// TwinCAT 3 PLC project DCSv1
// ProgramVersion: 3.1.4023.0
// libraries:
//   Tc2_MC2, * (Beckhoff Automation GmbH)
//   Tc2_MC2_Drive, * (Beckhoff Automation GmbH)
//   Tc2_SerialCom, * (Beckhoff Automation GmbH)
//   Tc2_Standard, * (Beckhoff Automation GmbH)
//   Tc2_System, * (Beckhoff Automation GmbH)
//   Tc2_Utilities, * (Beckhoff Automation GmbH)
//   Tc3_Module, * (Beckhoff Automation GmbH)
// project tree:
//   / ComTask.TcTTO, PlcTask.TcTTO
//   DUTs/DUTs/ arr8Bit.TcDUT
//   GVLs/GVLs/ GVL.TcGVL, GVL_IO.TcGVL (not stored), GVL_PN.TcGVL, GVL_RESD.TcGVL, GVL_ROB.TcGVL, ReadMe.TcGVL
//   POUs/Archive/ FB_Analog.TcPOU (not stored), P_ComEL6001.TcPOU (not stored)
//   POUs/Component/MIxer_Driver/ FB_Drive.TcPOU (not stored), FB_Mixer1_2.TcPOU
//   POUs/Component/ P_AP1_Check.TcPOU (not stored), P_AP1_OnOff.TcPOU (not stored), P_CC1_Enable.TcPOU (not stored), P_CP1_Check.TcPOU, P_CP1_Enable.TcPOU (not stored), P_MI1_OnOff.TcPOU (not stored), P_SP1_Check.TcPOU (not stored), P_SP1_OnOff.TcPOU (not stored)
//   POUs/Customed_Mode/ P_MI1_Curved_Speed.TcPOU (not stored)
//   POUs/ FB_GetOutputData.TcPOU, FB_Output_Speed.TcPOU (not stored), FB_SetConfigData.TcPOU (not stored), FB_SetOutputDataToIO.TcPOU, MAIN.TcPOU, P_Control_Mode.TcPOU, P_Manual_Operate.TcPOU (not stored), P_PNDataConvert.TcPOU, P_Robot_Operate.TcPOU, P_Laptop_Operate.TcPOU, temp.TcPOU
//   POUs/Utils/ F_Convert_2Byte_to_Uint.TcPOU, F_Convert_2Byte_to_Real.TcPOU, F_Convert_Bit_to_Byte.TcPOU, F_Convert_Uint_to_2Byte.TcPOU, F_LowpassFilter.TcPOU (not stored), F_Convert_2Byte_to_Int.TcPOU (not stored), F_Convert_Byte_to_Bit.TcPOU (not stored), F_Convert_Int_to_2Byte.TcPOU (not stored), F_DecimalData.TcPOU (not stored), F_Mapping.TcPOU (not stored), F_ScalAnalogOut.TcPOU
// real-time tasks:
//   TASK PlcTask: cycle T#10ms, priority 10, ADS port 350
//   TASK ComTask: cycle T#8ms, priority 5, ADS port 351
// motion (NC):
//   TASK NC-Task 1 SAF: cycle T#2ms, priority 4, ADS port 501
//   TASK NC-Task 1 SVB: cycle T#10ms, priority 8, ADS port 511
//   AXIS Mixer 1 (id 2)
//     General: UnitName=°, UnitFlags=#x00000004
//     Dynamic: Acceleration=7443.34, Deceleration=7443.34, Jerk=22330
//     Velo: RefSearch=49.6222741699219, RefSync=49.6222741699219, SlowManual=248.111370849609, FastManual=1488.66822509766, Fast=4962.22741699219, Maximum=4962.23
//     OtherSettings: AllowMotionCmdToSlave=true
//     encoder EncType=8
//       EncPara: ScaleFactorNumerator=45, ScaleFactorDenominator=1048576, Offset=-131121.7408, Inverse=true, MaxCount=#x007fffff, ReferenceSystem=2
//     drive DrvType=9
//       DrvPara: Inverse=true, MaxCount=#xffffffff, DriveControlDWord=#x00030100
//         Analog: VeloReferenz=5458.45015869141, VeloScale=1.02400649589962, ScaleFactorActTorque=0.1
//         TimeComp: TaskDelayCycles=1
//     controller CtrType=1
//       CtrPara: PriorControlFactor=1
//         Observer: BandWidth=20
//   AXIS Mixer 2 (id 3)
//     General: UnitName=°, UnitFlags=#x00000004
//     Dynamic: Acceleration=7443.34, Deceleration=7443.34, Jerk=22330
//     Velo: RefSearch=49.6222741699219, RefSync=49.6222741699219, SlowManual=248.111370849609, FastManual=1488.66822509766, Fast=4962.22741699219, Maximum=4962.23
//     OtherSettings: AllowMotionCmdToSlave=true
//     encoder EncType=8
//       EncPara: ScaleFactorNumerator=45, ScaleFactorDenominator=1048576, MaxCount=#x007fffff, ReferenceSystem=2
//     drive DrvType=9
//       DrvPara: MaxCount=#xffffffff, DriveControlDWord=#x00030100
//         Analog: VeloReferenz=5458.45015869141, VeloScale=1.02400649589962, ScaleFactorActTorque=0.1
//         TimeComp: TaskDelayCycles=1
//     controller CtrType=1
//       CtrPara: PriorControlFactor=1
//         Observer: BandWidth=20
// I/O:
//   DEVICE Device 1 (EtherCAT), AmsNetId 172.17.147.1.3.1
//     Term 1 (EK1200) [EK1200-5000 EtherCAT Power supply (2A E-Bus)]
//       Term 2 (EL1008) 30K3 [EL1008 8Ch. Dig. Input 24V, 3ms]
//       Term 3 (EL1008) 30K3.1 [EL1008 8Ch. Dig. Input 24V, 3ms]
//       Term 10 (EL1008) new [EL1008 8Ch. Dig. Input 24V, 3ms]
//       Term 4 (EL2008) 30K4 [EL2008 8Ch. Dig. Output 24V, 0.5A]
//       Term 5 (EL2008) 30K5 [EL2008 8Ch. Dig. Output 24V, 0.5A]
//       Term 12 (EL2008) new [EL2008 8Ch. Dig. Output 24V, 0.5A]
//       Term 13 (EL3022) new [EL3022 2Ch. Ana. Input 4-20mA DIFF]
//       Term 14 (EL3202) new [EL3202 2Ch. Ana. Input PT100 (RTD)]
//       Term 16 (EL3202) new pt100 [EL3202 2Ch. Ana. Input PT100 (RTD)]
//       Term 6 (EL3255) 30K5.1 [EL3255 5Ch. potentiometer measurement with sensor supply]
//       Term 7 (EL4134) 30K6 [EL4134 4Ch. Ana. Output -10/+10V, 16bit]
//       Term 8 (EL6001) [EL6001 Interface (RS232)]
//       Term 15 (EL6631-0010) [EL6631-0010 PROFINET IO Device]
//       Term 17 (EL6631) [EL6631 PROFINET IO Controller]
//       Term 9 (EL9011) [EL9011 End Terminal]
//   DEVICE Device 4 (EtherCAT), AmsNetId 172.17.147.1.5.1
//     Drive 11 (AX5206-0000-0213) [AX5206-0000-0213 EtherCAT Drive (SoE, 2 Ch.)]
//   DEVICE Device 1 (EL6631-0010), AmsNetId 5.57.158.168.2.1
//     robotbasicio [ABB Robotics The robot controller's internal PROFINET IO device. 888-3]
//       modules: Term 1 (DAP Module), Term 2 (DI 256 bytes), Term 3 (DO 256 bytes)
// variable links:
//   NC-Task 1 SAF/Axes/Mixer 1 <-> Device 4 (EtherCAT)/Drive 11 (AX5206-0000-0213)
//     Drive/Inputs/In/nDataIn1 <-> AT 1/Following distance
//     Drive/Inputs/In/nDcOutputTime <-> InfoData/DcOutputShift
//     Drive/Inputs/In/nState1 <-> AT 1/Drive status word @bit 8
//     Drive/Inputs/In/nState2 <-> AT 1/Drive status word
//     Drive/Inputs/In/nState4 @bit 1 <-> WcState/InputToggle
//     Drive/Inputs/In/nState4 <-> WcState/WcState
//     Drive/Outputs/Out/nCtrl1 <-> MDT 1/Master control word @bit 8
//     Drive/Outputs/Out/nDataOut1 <-> MDT 1/Position command value
//     Enc/Inputs/In/nDataIn1 <-> AT 1/Position feedback 1 value
//     Enc/Inputs/In/nDcInputTime <-> InfoData/DcInputShift
//     Enc/Inputs/In/nState4 @bit 1 <-> WcState/InputToggle
//     Enc/Inputs/In/nState4 <-> WcState/WcState
//   NC-Task 1 SAF/Axes/Mixer 2 <-> Device 4 (EtherCAT)/Drive 11 (AX5206-0000-0213)
//     Drive/Inputs/In/nDataIn1 <-> AT 2/Following distance
//     Drive/Inputs/In/nDcOutputTime <-> InfoData/DcOutputShift
//     Drive/Inputs/In/nState1 <-> AT 2/Drive status word @bit 8
//     Drive/Inputs/In/nState2 <-> AT 2/Drive status word
//     Drive/Inputs/In/nState4 @bit 1 <-> WcState/InputToggle
//     Drive/Inputs/In/nState4 <-> WcState/WcState
//     Drive/Outputs/Out/nCtrl1 <-> MDT 2/Master control word @bit 8
//     Drive/Outputs/Out/nDataOut1 <-> MDT 2/Position command value
//     Enc/Inputs/In/nDataIn1 <-> AT 2/Position feedback 1 value
//     Enc/Inputs/In/nDcInputTime <-> InfoData/DcInputShift
//     Enc/Inputs/In/nState4 @bit 1 <-> WcState/InputToggle
//     Enc/Inputs/In/nState4 <-> WcState/WcState
//   DCSv1/DCSv1 Instance <-> Device 1 (EL6631-0010)/robotbasicio
//     PlcTask Inputs/GVL_PN.DO_From_ROB <-> API/Term 3 (DO 256 bytes)/Subterm 5 (DO 256 bytes)/Inputs/Output 0
//     PlcTask Inputs/GVL_PN.DO_From_ROB[{0..4}] <-> API/Term 3 (DO 256 bytes)/Subterm 5 (DO 256 bytes)/Inputs/Output {0..4}  (5 links)
//     PlcTask Inputs/GVL_PN.GO_From_ROB[100] <-> API/Term 3 (DO 256 bytes)/Subterm 5 (DO 256 bytes)/Inputs/Output 100
//     PlcTask Inputs/GVL_PN.GO_From_ROB[101] <-> API/Term 3 (DO 256 bytes)/Subterm 5 (DO 256 bytes)/Inputs/Output 101
//     PlcTask Inputs/GVL_PN.GO_From_ROB[102] <-> API/Term 3 (DO 256 bytes)/Subterm 5 (DO 256 bytes)/Inputs/Output 102
//     PlcTask Inputs/GVL_PN.GO_From_ROB[103] <-> API/Term 3 (DO 256 bytes)/Subterm 5 (DO 256 bytes)/Inputs/Output 103
//     PlcTask Inputs/GVL_PN.GO_From_ROB[104] <-> API/Term 3 (DO 256 bytes)/Subterm 5 (DO 256 bytes)/Inputs/Output 104
//     PlcTask Inputs/GVL_PN.GO_From_ROB[105] <-> API/Term 3 (DO 256 bytes)/Subterm 5 (DO 256 bytes)/Inputs/Output 105
//     PlcTask Inputs/GVL_PN.GO_From_ROB[32] <-> API/Term 3 (DO 256 bytes)/Subterm 5 (DO 256 bytes)/Inputs/Output 32
//     PlcTask Inputs/GVL_PN.GO_From_ROB[33] <-> API/Term 3 (DO 256 bytes)/Subterm 5 (DO 256 bytes)/Inputs/Output 33
//     PlcTask Inputs/GVL_PN.GO_From_ROB[47] <-> API/Term 3 (DO 256 bytes)/Subterm 5 (DO 256 bytes)/Inputs/Output 47
//     PlcTask Inputs/GVL_PN.GO_From_ROB[48] <-> API/Term 3 (DO 256 bytes)/Subterm 5 (DO 256 bytes)/Inputs/Output 48
//     PlcTask Inputs/GVL_PN.GO_From_ROB[62] <-> API/Term 3 (DO 256 bytes)/Subterm 5 (DO 256 bytes)/Inputs/Output 62
//     PlcTask Inputs/GVL_PN.GO_From_ROB[63] <-> API/Term 3 (DO 256 bytes)/Subterm 5 (DO 256 bytes)/Inputs/Output 63
//     PlcTask Inputs/GVL_PN.GO_From_ROB[64] <-> API/Term 3 (DO 256 bytes)/Subterm 5 (DO 256 bytes)/Inputs/Output 64
//     PlcTask Inputs/GVL_PN.GO_From_ROB[65] <-> API/Term 3 (DO 256 bytes)/Subterm 5 (DO 256 bytes)/Inputs/Output 65
//     PlcTask Inputs/GVL_PN.GO_From_ROB[66] <-> API/Term 3 (DO 256 bytes)/Subterm 5 (DO 256 bytes)/Inputs/Output 66
//     PlcTask Inputs/GVL_PN.GO_From_ROB[67] <-> API/Term 3 (DO 256 bytes)/Subterm 5 (DO 256 bytes)/Inputs/Output 67
//     PlcTask Inputs/GVL_PN.GO_From_ROB[68] <-> API/Term 3 (DO 256 bytes)/Subterm 5 (DO 256 bytes)/Inputs/Output 68
//     PlcTask Inputs/GVL_PN.GO_From_ROB[69] <-> API/Term 3 (DO 256 bytes)/Subterm 5 (DO 256 bytes)/Inputs/Output 69
//     PlcTask Inputs/GVL_PN.GO_From_ROB[70] <-> API/Term 3 (DO 256 bytes)/Subterm 5 (DO 256 bytes)/Inputs/Output 70
//     PlcTask Inputs/GVL_PN.GO_From_ROB[71] <-> API/Term 3 (DO 256 bytes)/Subterm 5 (DO 256 bytes)/Inputs/Output 71
//     PlcTask Inputs/GVL_PN.GO_From_ROB[72] <-> API/Term 3 (DO 256 bytes)/Subterm 5 (DO 256 bytes)/Inputs/Output 72
//     PlcTask Inputs/GVL_PN.GO_From_ROB[73] <-> API/Term 3 (DO 256 bytes)/Subterm 5 (DO 256 bytes)/Inputs/Output 73
//     PlcTask Inputs/GVL_PN.GO_From_ROB[74] <-> API/Term 3 (DO 256 bytes)/Subterm 5 (DO 256 bytes)/Inputs/Output 74
//     PlcTask Inputs/GVL_PN.GO_From_ROB[75] <-> API/Term 3 (DO 256 bytes)/Subterm 5 (DO 256 bytes)/Inputs/Output 75
//     PlcTask Inputs/GVL_PN.GO_From_ROB[78] <-> API/Term 3 (DO 256 bytes)/Subterm 5 (DO 256 bytes)/Inputs/Output 78
//     PlcTask Inputs/GVL_PN.GO_From_ROB[79] <-> API/Term 3 (DO 256 bytes)/Subterm 5 (DO 256 bytes)/Inputs/Output 79
//     PlcTask Inputs/GVL_PN.GO_From_ROB[80] <-> API/Term 3 (DO 256 bytes)/Subterm 5 (DO 256 bytes)/Inputs/Output 80
//     PlcTask Inputs/GVL_PN.GO_From_ROB[81] <-> API/Term 3 (DO 256 bytes)/Subterm 5 (DO 256 bytes)/Inputs/Output 81
//     PlcTask Inputs/GVL_PN.GO_From_ROB[82] <-> API/Term 3 (DO 256 bytes)/Subterm 5 (DO 256 bytes)/Inputs/Output 82
//     PlcTask Inputs/GVL_PN.GO_From_ROB[83] <-> API/Term 3 (DO 256 bytes)/Subterm 5 (DO 256 bytes)/Inputs/Output 83
//     PlcTask Inputs/GVL_PN.GO_From_ROB[84] <-> API/Term 3 (DO 256 bytes)/Subterm 5 (DO 256 bytes)/Inputs/Output 84
//     PlcTask Inputs/GVL_PN.GO_From_ROB[85] <-> API/Term 3 (DO 256 bytes)/Subterm 5 (DO 256 bytes)/Inputs/Output 85
//     PlcTask Inputs/GVL_PN.GO_From_ROB[86] <-> API/Term 3 (DO 256 bytes)/Subterm 5 (DO 256 bytes)/Inputs/Output 86
//     PlcTask Inputs/GVL_PN.GO_From_ROB[87] <-> API/Term 3 (DO 256 bytes)/Subterm 5 (DO 256 bytes)/Inputs/Output 87
//     PlcTask Inputs/GVL_PN.GO_From_ROB[88] <-> API/Term 3 (DO 256 bytes)/Subterm 5 (DO 256 bytes)/Inputs/Output 88
//     PlcTask Inputs/GVL_PN.GO_From_ROB[89] <-> API/Term 3 (DO 256 bytes)/Subterm 5 (DO 256 bytes)/Inputs/Output 89
//     PlcTask Inputs/GVL_PN.GO_From_ROB[90] <-> API/Term 3 (DO 256 bytes)/Subterm 5 (DO 256 bytes)/Inputs/Output 90
//     PlcTask Inputs/GVL_PN.GO_From_ROB[91] <-> API/Term 3 (DO 256 bytes)/Subterm 5 (DO 256 bytes)/Inputs/Output 91
//     PlcTask Inputs/GVL_PN.GO_From_ROB[94] <-> API/Term 3 (DO 256 bytes)/Subterm 5 (DO 256 bytes)/Inputs/Output 94
//     PlcTask Inputs/GVL_PN.GO_From_ROB[95] <-> API/Term 3 (DO 256 bytes)/Subterm 5 (DO 256 bytes)/Inputs/Output 95
//     PlcTask Inputs/GVL_PN.GO_From_ROB[96] <-> API/Term 3 (DO 256 bytes)/Subterm 5 (DO 256 bytes)/Inputs/Output 96
//     PlcTask Inputs/GVL_PN.GO_From_ROB[97] <-> API/Term 3 (DO 256 bytes)/Subterm 5 (DO 256 bytes)/Inputs/Output 97
//     PlcTask Inputs/GVL_PN.GO_From_ROB[98] <-> API/Term 3 (DO 256 bytes)/Subterm 5 (DO 256 bytes)/Inputs/Output 98
//     PlcTask Inputs/GVL_PN.GO_From_ROB[99] <-> API/Term 3 (DO 256 bytes)/Subterm 5 (DO 256 bytes)/Inputs/Output 99
//     PlcTask Outputs/GVL_PN.DI_To_ROB[0]/data8Bit[0] <-> API/Term 2 (DI 256 bytes)/Subterm 4 (DI 256 bytes)/Outputs/Input 0[0]
//     PlcTask Outputs/GVL_PN.DI_To_ROB[0]/data8Bit[1] <-> API/Term 2 (DI 256 bytes)/Subterm 4 (DI 256 bytes)/Outputs/Input 0[1]
//     PlcTask Outputs/GVL_PN.DI_To_ROB[0]/data8Bit[2] <-> API/Term 2 (DI 256 bytes)/Subterm 4 (DI 256 bytes)/Outputs/Input 0[2]
//     PlcTask Outputs/GVL_PN.DI_To_ROB[0]/data8Bit[3] <-> API/Term 2 (DI 256 bytes)/Subterm 4 (DI 256 bytes)/Outputs/Input 0[3]
//     PlcTask Outputs/GVL_PN.DI_To_ROB[0]/data8Bit[4] <-> API/Term 2 (DI 256 bytes)/Subterm 4 (DI 256 bytes)/Outputs/Input 0[4]
//     PlcTask Outputs/GVL_PN.DI_To_ROB[0]/data8Bit[5] <-> API/Term 2 (DI 256 bytes)/Subterm 4 (DI 256 bytes)/Outputs/Input 0[5]
//     PlcTask Outputs/GVL_PN.DI_To_ROB[0]/data8Bit[6] <-> API/Term 2 (DI 256 bytes)/Subterm 4 (DI 256 bytes)/Outputs/Input 0[6]
//     PlcTask Outputs/GVL_PN.DI_To_ROB[0]/data8Bit[7] <-> API/Term 2 (DI 256 bytes)/Subterm 4 (DI 256 bytes)/Outputs/Input 0[7]
//     PlcTask Outputs/GVL_PN.DI_To_ROB[1]/data8Bit[0] <-> API/Term 2 (DI 256 bytes)/Subterm 4 (DI 256 bytes)/Outputs/Input 1[0]
//     PlcTask Outputs/GVL_PN.DI_To_ROB[1]/data8Bit[1] <-> API/Term 2 (DI 256 bytes)/Subterm 4 (DI 256 bytes)/Outputs/Input 1[1]
//     PlcTask Outputs/GVL_PN.DI_To_ROB[1]/data8Bit[2] <-> API/Term 2 (DI 256 bytes)/Subterm 4 (DI 256 bytes)/Outputs/Input 1[2]
//     PlcTask Outputs/GVL_PN.DI_To_ROB[1]/data8Bit[3] <-> API/Term 2 (DI 256 bytes)/Subterm 4 (DI 256 bytes)/Outputs/Input 1[3]
//     PlcTask Outputs/GVL_PN.DI_To_ROB[1]/data8Bit[4] <-> API/Term 2 (DI 256 bytes)/Subterm 4 (DI 256 bytes)/Outputs/Input 1[4]
//     PlcTask Outputs/GVL_PN.DI_To_ROB[1]/data8Bit[5] <-> API/Term 2 (DI 256 bytes)/Subterm 4 (DI 256 bytes)/Outputs/Input 1[5]
//     PlcTask Outputs/GVL_PN.DI_To_ROB[1]/data8Bit[6] <-> API/Term 2 (DI 256 bytes)/Subterm 4 (DI 256 bytes)/Outputs/Input 1[6]
//     PlcTask Outputs/GVL_PN.DI_To_ROB[1]/data8Bit[7] <-> API/Term 2 (DI 256 bytes)/Subterm 4 (DI 256 bytes)/Outputs/Input 1[7]
//     PlcTask Outputs/GVL_PN.DI_To_ROB[2]/data8Bit[0] <-> API/Term 2 (DI 256 bytes)/Subterm 4 (DI 256 bytes)/Outputs/Input 2[0]
//     PlcTask Outputs/GVL_PN.DI_To_ROB[2]/data8Bit[1] <-> API/Term 2 (DI 256 bytes)/Subterm 4 (DI 256 bytes)/Outputs/Input 2[1]
//     PlcTask Outputs/GVL_PN.DI_To_ROB[2]/data8Bit[2] <-> API/Term 2 (DI 256 bytes)/Subterm 4 (DI 256 bytes)/Outputs/Input 2[2]
//     PlcTask Outputs/GVL_PN.DI_To_ROB[2]/data8Bit[3] <-> API/Term 2 (DI 256 bytes)/Subterm 4 (DI 256 bytes)/Outputs/Input 2[3]
//     PlcTask Outputs/GVL_PN.DI_To_ROB[2]/data8Bit[4] <-> API/Term 2 (DI 256 bytes)/Subterm 4 (DI 256 bytes)/Outputs/Input 2[4]
//     PlcTask Outputs/GVL_PN.DI_To_ROB[2]/data8Bit[5] <-> API/Term 2 (DI 256 bytes)/Subterm 4 (DI 256 bytes)/Outputs/Input 2[5]
//     PlcTask Outputs/GVL_PN.DI_To_ROB[2]/data8Bit[6] <-> API/Term 2 (DI 256 bytes)/Subterm 4 (DI 256 bytes)/Outputs/Input 2[6]
//     PlcTask Outputs/GVL_PN.DI_To_ROB[2]/data8Bit[7] <-> API/Term 2 (DI 256 bytes)/Subterm 4 (DI 256 bytes)/Outputs/Input 2[7]
//     PlcTask Outputs/GVL_PN.DI_To_ROB[3]/data8Bit[0] <-> API/Term 2 (DI 256 bytes)/Subterm 4 (DI 256 bytes)/Outputs/Input 3[0]
//     PlcTask Outputs/GVL_PN.DI_To_ROB[3]/data8Bit[1] <-> API/Term 2 (DI 256 bytes)/Subterm 4 (DI 256 bytes)/Outputs/Input 3[1]
//     PlcTask Outputs/GVL_PN.DI_To_ROB[3]/data8Bit[2] <-> API/Term 2 (DI 256 bytes)/Subterm 4 (DI 256 bytes)/Outputs/Input 3[2]
//     PlcTask Outputs/GVL_PN.DI_To_ROB[3]/data8Bit[3] <-> API/Term 2 (DI 256 bytes)/Subterm 4 (DI 256 bytes)/Outputs/Input 3[3]
//     PlcTask Outputs/GVL_PN.DI_To_ROB[3]/data8Bit[4] <-> API/Term 2 (DI 256 bytes)/Subterm 4 (DI 256 bytes)/Outputs/Input 3[4]
//     PlcTask Outputs/GVL_PN.DI_To_ROB[3]/data8Bit[5] <-> API/Term 2 (DI 256 bytes)/Subterm 4 (DI 256 bytes)/Outputs/Input 3[5]
//     PlcTask Outputs/GVL_PN.DI_To_ROB[3]/data8Bit[6] <-> API/Term 2 (DI 256 bytes)/Subterm 4 (DI 256 bytes)/Outputs/Input 3[6]
//     PlcTask Outputs/GVL_PN.DI_To_ROB[3]/data8Bit[7] <-> API/Term 2 (DI 256 bytes)/Subterm 4 (DI 256 bytes)/Outputs/Input 3[7]
//     PlcTask Outputs/GVL_PN.DI_To_ROB[4]/data8Bit[0] <-> API/Term 2 (DI 256 bytes)/Subterm 4 (DI 256 bytes)/Outputs/Input 4[0]
//     PlcTask Outputs/GVL_PN.DI_To_ROB[4]/data8Bit[1] <-> API/Term 2 (DI 256 bytes)/Subterm 4 (DI 256 bytes)/Outputs/Input 4[1]
//     PlcTask Outputs/GVL_PN.DI_To_ROB[4]/data8Bit[2] <-> API/Term 2 (DI 256 bytes)/Subterm 4 (DI 256 bytes)/Outputs/Input 4[2]
//     PlcTask Outputs/GVL_PN.DI_To_ROB[4]/data8Bit[3] <-> API/Term 2 (DI 256 bytes)/Subterm 4 (DI 256 bytes)/Outputs/Input 4[3]
//     PlcTask Outputs/GVL_PN.DI_To_ROB[4]/data8Bit[4] <-> API/Term 2 (DI 256 bytes)/Subterm 4 (DI 256 bytes)/Outputs/Input 4[4]
//     PlcTask Outputs/GVL_PN.DI_To_ROB[4]/data8Bit[5] <-> API/Term 2 (DI 256 bytes)/Subterm 4 (DI 256 bytes)/Outputs/Input 4[5]
//     PlcTask Outputs/GVL_PN.DI_To_ROB[4]/data8Bit[6] <-> API/Term 2 (DI 256 bytes)/Subterm 4 (DI 256 bytes)/Outputs/Input 4[6]
//     PlcTask Outputs/GVL_PN.DI_To_ROB[4]/data8Bit[7] <-> API/Term 2 (DI 256 bytes)/Subterm 4 (DI 256 bytes)/Outputs/Input 4[7]
//     PlcTask Outputs/GVL_PN.GI_To_ROB[106] <-> API/Term 2 (DI 256 bytes)/Subterm 4 (DI 256 bytes)/Outputs/Input 106
//     PlcTask Outputs/GVL_PN.GI_To_ROB[107] <-> API/Term 2 (DI 256 bytes)/Subterm 4 (DI 256 bytes)/Outputs/Input 107
//     PlcTask Outputs/GVL_PN.GI_To_ROB[32] <-> API/Term 2 (DI 256 bytes)/Subterm 4 (DI 256 bytes)/Outputs/Input 32
//     PlcTask Outputs/GVL_PN.GI_To_ROB[33] <-> API/Term 2 (DI 256 bytes)/Subterm 4 (DI 256 bytes)/Outputs/Input 33
//     PlcTask Outputs/GVL_PN.GI_To_ROB[47] <-> API/Term 2 (DI 256 bytes)/Subterm 4 (DI 256 bytes)/Outputs/Input 47
//     PlcTask Outputs/GVL_PN.GI_To_ROB[48] <-> API/Term 2 (DI 256 bytes)/Subterm 4 (DI 256 bytes)/Outputs/Input 48
//     PlcTask Outputs/GVL_PN.GI_To_ROB[49] <-> API/Term 2 (DI 256 bytes)/Subterm 4 (DI 256 bytes)/Outputs/Input 49
//     PlcTask Outputs/GVL_PN.GI_To_ROB[50] <-> API/Term 2 (DI 256 bytes)/Subterm 4 (DI 256 bytes)/Outputs/Input 50
//     PlcTask Outputs/GVL_PN.GI_To_ROB[51] <-> API/Term 2 (DI 256 bytes)/Subterm 4 (DI 256 bytes)/Outputs/Input 51
//     PlcTask Outputs/GVL_PN.GI_To_ROB[52] <-> API/Term 2 (DI 256 bytes)/Subterm 4 (DI 256 bytes)/Outputs/Input 52
//     PlcTask Outputs/GVL_PN.GI_To_ROB[53] <-> API/Term 2 (DI 256 bytes)/Subterm 4 (DI 256 bytes)/Outputs/Input 53
//     PlcTask Outputs/GVL_PN.GI_To_ROB[54] <-> API/Term 2 (DI 256 bytes)/Subterm 4 (DI 256 bytes)/Outputs/Input 54
//     PlcTask Outputs/GVL_PN.GI_To_ROB[55] <-> API/Term 2 (DI 256 bytes)/Subterm 4 (DI 256 bytes)/Outputs/Input 55
//     PlcTask Outputs/GVL_PN.GI_To_ROB[56] <-> API/Term 2 (DI 256 bytes)/Subterm 4 (DI 256 bytes)/Outputs/Input 56
//     PlcTask Outputs/GVL_PN.GI_To_ROB[57] <-> API/Term 2 (DI 256 bytes)/Subterm 4 (DI 256 bytes)/Outputs/Input 57
//     PlcTask Outputs/GVL_PN.GI_To_ROB[58] <-> API/Term 2 (DI 256 bytes)/Subterm 4 (DI 256 bytes)/Outputs/Input 58
//     PlcTask Outputs/GVL_PN.GI_To_ROB[59] <-> API/Term 2 (DI 256 bytes)/Subterm 4 (DI 256 bytes)/Outputs/Input 59
//     PlcTask Outputs/GVL_PN.GI_To_ROB[60] <-> API/Term 2 (DI 256 bytes)/Subterm 4 (DI 256 bytes)/Outputs/Input 60
//     PlcTask Outputs/GVL_PN.GI_To_ROB[61] <-> API/Term 2 (DI 256 bytes)/Subterm 4 (DI 256 bytes)/Outputs/Input 61
//     PlcTask Outputs/GVL_PN.GI_To_ROB[62] <-> API/Term 2 (DI 256 bytes)/Subterm 4 (DI 256 bytes)/Outputs/Input 62
//     PlcTask Outputs/GVL_PN.GI_To_ROB[77] <-> API/Term 2 (DI 256 bytes)/Subterm 4 (DI 256 bytes)/Outputs/Input 77
//     PlcTask Outputs/GVL_PN.GI_To_ROB[78] <-> API/Term 2 (DI 256 bytes)/Subterm 4 (DI 256 bytes)/Outputs/Input 78
//     PlcTask Outputs/GVL_PN.GI_To_ROB[79] <-> API/Term 2 (DI 256 bytes)/Subterm 4 (DI 256 bytes)/Outputs/Input 79
//     PlcTask Outputs/GVL_PN.GI_To_ROB[80] <-> API/Term 2 (DI 256 bytes)/Subterm 4 (DI 256 bytes)/Outputs/Input 80
//     PlcTask Outputs/GVL_PN.GI_To_ROB[81] <-> API/Term 2 (DI 256 bytes)/Subterm 4 (DI 256 bytes)/Outputs/Input 81
//     PlcTask Outputs/GVL_PN.GI_To_ROB[82] <-> API/Term 2 (DI 256 bytes)/Subterm 4 (DI 256 bytes)/Outputs/Input 82
//     PlcTask Outputs/GVL_PN.GI_To_ROB[92] <-> API/Term 2 (DI 256 bytes)/Subterm 4 (DI 256 bytes)/Outputs/Input 92
//     PlcTask Outputs/GVL_PN.GI_To_ROB[93] <-> API/Term 2 (DI 256 bytes)/Subterm 4 (DI 256 bytes)/Outputs/Input 93
//   DCSv1/DCSv1 Instance <-> Device 1 (EtherCAT)/Term 1 (EK1200)/Term 10 (EL1008) new
//     PlcTask Inputs/GVL_IO.ib_SP1_No_Error <-> Channel 2/Input
//     PlcTask Inputs/GVL_IO.ib_SP1_Ready <-> Channel 1/Input
//   DCSv1/DCSv1 Instance <-> Device 1 (EtherCAT)/Term 1 (EK1200)/Term 13 (EL3022) new
//     PlcTask Inputs/GVL_IO.in_Pressure_Funnel <-> AI Standard Channel 1/Value
//     PlcTask Inputs/GVL_IO.in_Pressure_Pump <-> AI Standard Channel 2/Value
//   DCSv1/DCSv1 Instance <-> Device 1 (EtherCAT)/Term 1 (EK1200)/Term 14 (EL3202) new
//     PlcTask Inputs/GVL_IO.in_Temp_CPump <-> RTD Inputs Channel 2/Value
//     PlcTask Inputs/GVL_IO.in_Temp_CPump_fresh <-> RTD Inputs Channel 1/Value
//   DCSv1/DCSv1 Instance <-> Device 1 (EtherCAT)/Term 1 (EK1200)/Term 16 (EL3202) new pt100
//     PlcTask Inputs/GVL_IO.in_Temp_Funnel_Outlet <-> RTD Inputs Channel 2/Value
//   DCSv1/DCSv1 Instance <-> Device 1 (EtherCAT)/Term 1 (EK1200)/Term 2 (EL1008) 30K3
//     PlcTask Inputs/GVL_IO.ib_AP1_No_Error <-> Channel 6/Input
//     PlcTask Inputs/GVL_IO.ib_AP1_Ready <-> Channel 5/Input
//     PlcTask Inputs/GVL_IO.ib_CC1_Button_Mode_Laptop <-> Channel 8/Input
//     PlcTask Inputs/GVL_IO.ib_CC1_Button_Reset <-> Channel 7/Input
//     PlcTask Inputs/GVL_IO.ib_CC1_Safety_Ready <-> Channel 1/Input
//     PlcTask Inputs/GVL_IO.ib_CP1_Drive_Error <-> Channel 4/Input
//     PlcTask Inputs/GVL_IO.ib_CP1_Ready <-> Channel 3/Input
//     PlcTask Inputs/GVL_IO.ib_CP1_Safety_Grid_Mounted <-> Channel 2/Input
//   DCSv1/DCSv1 Instance <-> Device 1 (EtherCAT)/Term 1 (EK1200)/Term 3 (EL1008) 30K3.1
//     PlcTask Inputs/GVL_IO.ib_AP1_Button_Not_Off <-> Channel 7/Input
//     PlcTask Inputs/GVL_IO.ib_AP1_Button_On <-> Channel 6/Input
//     PlcTask Inputs/GVL_IO.ib_CC1_Button_Mode_Manual <-> Channel 1/Input
//     PlcTask Inputs/GVL_IO.ib_MI1_Button_Not_Off <-> Channel 3/Input
//     PlcTask Inputs/GVL_IO.ib_MI1_Button_On <-> Channel 2/Input
//     PlcTask Inputs/GVL_IO.ib_SP1_Button_Not_Off <-> Channel 5/Input
//     PlcTask Inputs/GVL_IO.ib_SP1_Button_On <-> Channel 4/Input
//   DCSv1/DCSv1 Instance <-> Device 1 (EtherCAT)/Term 1 (EK1200)/Term 4 (EL2008) 30K4
//     PlcTask Outputs/GVL_IO.ob_AP1_Pressure_Ok <-> Channel 7/Output
//     PlcTask Outputs/GVL_IO.ob_AP1_Pulse <-> Channel 8/Output
//     PlcTask Outputs/GVL_IO.ob_AP1_Start <-> Channel 6/Output
//     PlcTask Outputs/GVL_IO.ob_CC1_Safety_Reset <-> Channel 1/Output
//     PlcTask Outputs/GVL_IO.ob_CP1_Backward <-> Channel 5/Output
//     PlcTask Outputs/GVL_IO.ob_CP1_Forward <-> Channel 4/Output
//     PlcTask Outputs/GVL_IO.ob_CP1_Start <-> Channel 3/Output
//     PlcTask Outputs/GVL_IO.ob_CP1_Stop <-> Channel 2/Output
//   DCSv1/DCSv1 Instance <-> Device 1 (EtherCAT)/Term 1 (EK1200)/Term 5 (EL2008) 30K5
//     PlcTask Outputs/GVL_IO.ob_AP1_Not_Empty <-> Channel 1/Output
//     PlcTask Outputs/GVL_IO.ob_AP1_Power_On <-> Channel 2/Output
//     PlcTask Outputs/GVL_IO.ob_SP1_Not_Empty <-> Channel 6/Output
//     PlcTask Outputs/GVL_IO.ob_SP1_Power_On <-> Channel 7/Output
//     PlcTask Outputs/GVL_IO.ob_SP1_Pressure_Ok <-> Channel 4/Output
//     PlcTask Outputs/GVL_IO.ob_SP1_Pulse <-> Channel 5/Output
//     PlcTask Outputs/GVL_IO.ob_SP1_Start <-> Channel 3/Output
//   DCSv1/DCSv1 Instance <-> Device 1 (EtherCAT)/Term 1 (EK1200)/Term 6 (EL3255) 30K5.1
//     PlcTask Inputs/GVL.nInputSpare1 <-> AI Standard Channel 4/Value
//     PlcTask Inputs/GVL.nInputSpare2 <-> AI Standard Channel 5/Value
//     PlcTask Inputs/GVL_IO.in_AP1_Poti_Speed <-> AI Standard Channel 3/Value
//     PlcTask Inputs/GVL_IO.in_MI1_Poti_Speed <-> AI Standard Channel 1/Value
//   DCSv1/DCSv1 Instance <-> Device 1 (EtherCAT)/Term 1 (EK1200)/Term 7 (EL4134) 30K6
//     PlcTask Outputs/GVL_IO.on_AP1_Speed <-> AO Output Channel 2/Analog output
//     PlcTask Outputs/GVL_IO.on_CP1_Speed <-> AO Output Channel 1/Analog output
//     PlcTask Outputs/GVL_IO.on_SP1_Speed <-> AO Output Channel 3/Analog output
//   DCSv1/DCSv1 Instance <-> Device 1 (EtherCAT)/Term 1 (EK1200)/Term 8 (EL6001)
//     ComTask Inputs/GVL.stIn_EL6001/D <-> COM Inputs/Data In 0
//     ComTask Inputs/GVL.stIn_EL6001/D @bit {8..168 step 8} <-> COM Inputs/Data In {1..21}  (21 links)
//     ComTask Inputs/GVL.stIn_EL6001/Status <-> COM Inputs/Status
//     ComTask Outputs/GVL.stOut_EL6001/Ctrl <-> COM Outputs/Ctrl
//     ComTask Outputs/GVL.stOut_EL6001/D <-> COM Outputs/Data Out 0
//     ComTask Outputs/GVL.stOut_EL6001/D @bit {8..168 step 8} <-> COM Outputs/Data Out {1..21}  (21 links)
//   DCSv1/DCSv1 Instance <-> Device 4 (EtherCAT)/Drive 11 (AX5206-0000-0213)
//     PlcTask Inputs/GVL_IO.in_MID1_ActAbsCurrent <-> AT 1/Actual absolute current
//     PlcTask Inputs/GVL_IO.in_MID2_ActAbsCurrent <-> AT 2/Actual absolute current
//     PlcTask Inputs/GVL_IO.in_MID1_ActMotorTemperature <-> AT 1/Motor temperature
//     PlcTask Inputs/GVL_IO.in_MID2_ActMotorTemperature <-> AT 2/Motor temperature
//   DCSv1/DCSv1 Instance <-> NC-Task 1 SAF/Axes/Mixer 1
//     PlcTask Inputs/GVL.Axis_Mixer1.NcToPlc <-> Outputs/ToPlc
//     PlcTask Outputs/GVL.Axis_Mixer1.PlcToNc <-> Inputs/FromPlc
//   DCSv1/DCSv1 Instance <-> NC-Task 1 SAF/Axes/Mixer 2
//     PlcTask Inputs/GVL.Axis_Mixer2.NcToPlc <-> Outputs/ToPlc
//     PlcTask Outputs/GVL.Axis_Mixer2.PlcToNc <-> Inputs/FromPlc

CONFIGURATION DCSv1
    RESOURCE PLC ON TwinCAT3
        TASK ComTask(INTERVAL := T#8ms, PRIORITY := 5);
        TASK PlcTask(INTERVAL := T#10ms, PRIORITY := 10);
        PROGRAM P_ComEL6001 WITH ComTask : P_ComEL6001;
        PROGRAM MAIN WITH PlcTask : MAIN;
    END_RESOURCE
END_CONFIGURATION

// ---- DUTs/DUTs/arr8Bit.TcDUT
TYPE arr8Bit :
STRUCT
	data8Bit : ARRAY[0..7] OF BOOL;
END_STRUCT
END_TYPE

// ---- GVLs/GVLs/GVL.TcGVL
{attribute 'qualified_only'}
// ***********************************************************************************
//
// Müller-steinag Gruppe, Kandergrien Einigen, CH-3646 Bern
// ETH Zurich, Building HIF E26, Laura-Hezner-Weg 7, CH-8093 Zürich
// 
// ***********************************************************************************
// 
// PROJECT     :  A061 Digital Casting System 
// FUNCTION    :  Global Varable Decelerate
// AUTHOR      :  Weiting Chen
// EMAIL       :  chenw@usi.ch
// Copyright   :  USI Mendrisio; ETH Zürich; Müller-steinag Gruppe (CH) 2023
// Contributor :  Mathias Suter/ Philippe Fleischmann
//
// ***********************************************************************************

VAR_GLOBAL
	
    // get
	//
	// Concrete Controller 1
	b_mode_manual : BOOL;
	b_mode_laptop : BOOL; 
	b_mode_robot : BOOL;  
	
	b_CC1_enable :BOOL;
	b_CC1_power_on: BOOL;
	s_current_mode: STRING;
	
	//
	// Mixer 1
	b_MI1_ReadToDrive : BOOL;
	b_MI1_Is_Run : BOOL;
	
	f_MI1_MaxSpeed : REAL := 720 ; //distance/s] (equel to 120 rpm, by measurement 221006)
	n_MI1_OverrideSpeed :INT;
	b_Ml1_Enable : BOOL;
	b_Ml1_Set_Run : BOOL;
	
	f_MI1_ActSpeedM1 : INT;
	f_MI1_ActSpeedM2 : INT;
	
	// Data Communication Axis Mixers
	// Mixer drive A 
	Axis_Mixer1: AXIS_REF;
	
	f_MID1_ActCurrent:REAL;
	f_MID1_ActTorque:REAL;
	
	//
	// Mixer drive B
	Axis_Mixer2: AXIS_REF;
	f_MID2_ActCurrent:REAL;
	f_MID2_ActTorque:REAL;
	
	//
	// Concrete Pump 1
	b_CP1_Check_On : BOOL; //??
	b_CP1_is_run : BOOL;
	b_CP1_is_ready : BOOL;	
	b_CP1_power_on :BOOL;
	b_CP1_safety_grid_on : BOOL;
	b_CP1_drive_error :BOOL;
	
	//
	// Admixture pump 1 (High dosage)
	b_AP1_Is_Run : BOOL;
	b_AP1_Check_On : BOOL;
	b_AP1_is_ready : BOOL;
	b_AP1_no_error : BOOL;
	
	//f_AP1_Override : LREAL; 
	
	//
	// Spare Admixture pump 1 (Low dosage)
	b_SP1_Is_Run : BOOL;
	b_SP1_Check_On : BOOL;
	b_SP1_is_ready : BOOL;
	b_SP1_no_error : BOOL;
	
	//f_SP1_Override :LREAL;

	// Config
	// Concrete Pump 1
	f_CP1_Max_Flowrate : REAL;
	f_CP1_Check_Flowrate : REAL;
	t_CP1_Check_Duration : TIME;
 	n_CP1_Flush_Flowrate :REAL;
	
	// Admixture pump (High)
	n_AP1_Max_Flowrate : REAL;
	n_AP1_Check_Flowrate : REAL;
	t_AP1_Check_Duration : TIME;
	n_AP1_Flush_Flowrate : REAL;
	f_AP1_Check_Mass : REAL;
	
	// Admixture pump (low)
	n_SP1_Max_Flowrate : REAL;
	n_SP1_Check_Flowrate : REAL;
	t_SP1_Check_Duration : TIME;
	n_SP1_Flush_Flowrate : REAL;
	f_SP1_Check_Mass : REAL;
	
	
	
	
	
	// 
	// Data Communication RS-232 (Spare)
	TxBufferEL								: ComBuffer;
	RxBufferEL								: ComBuffer;
	
			

	//
	// Control Input Speed
	fControlMixerPumpSpeed					: REAL; 
	fControlPeristalticPumpSpeed			: REAL; 
	fControlDosingPumpSpeed					: REAL; 
	fInputSpare1							: REAL; 
	fInputSpare2							: REAL; 
	
	//
	// Output Speed
	fConcretePumpSpeed						: REAL;
	fDosingPumpSpeed						: REAL;
	fOutputSpare1							: REAL;
	fOutputSpare2							: REAL;
	
	
	//
	//Hardware Input
	bSafetyIO						AT %I*	: BOOL;
	// bConcretePumpSafetyGridMounted	AT %I*	: BOOL;
	// bConcretePumpReady				AT %I*	: BOOL;
	// bConcretePumpFcError				AT %I*	: BOOL;
	bDosingPumpReady				AT %I*	: BOOL;
	bDosingPumpNoError				AT %I*	: BOOL;
	bControlResetSafety				AT %I*	: BOOL;
	bControlLaptop					AT %I*	: BOOL;
	bControlManual					AT %I*	: BOOL;	
	nControlMixerPumpOn				AT %I*	: BOOL; 
	nControlMixerPumpOff			AT %I*	: BOOL; 
	nControlConcretPumpOn			AT %I*	: BOOL; 
	nControlConcretPumpOff			AT %I*	: BOOL; 
	nControlDosingPumpOn			AT %I*	: BOOL; 
	nControlDosingPumpOff			AT %I*	: BOOL; 
	bInputSpare1					AT %I*	: BOOL;
		
	nControlMixerPumpSpeed			AT %I*	: INT; 
	// nControlPeristalticPumpSpeed	AT %I*	: INT; 
	nControlDosingPumpSpeed			AT %I*	: INT; 
	nInputSpare1					AT %I*	: INT; 
	nInputSpare2					AT %I*	: INT; 

	
	//
	//Hardware Output
	bResetSafety					AT %Q*	: BOOL;
	// bConcretePumpOn					AT %Q*	: BOOL;
	// bConcretePumpOff					AT %Q*	: BOOL;
	// bConcretePumpForwardOn			AT %Q*	: BOOL;
	// bConcretePumpBackwardOn			AT %Q*	: BOOL;
	bDosingPumpDosingHighLow		AT %Q*	: BOOL;
	bDosingPumpNoFastStop			AT %Q*	: BOOL;
	bDosingPumpDosingAmount			AT %Q*	: BOOL;
	bOutputSpare1					AT %Q*	: BOOL;
	bOutputSpare2					AT %Q*	: BOOL;
	bOutputSpare3					AT %Q*	: BOOL;
	bOutputSpare4					AT %Q*	: BOOL;
	bOutputSpare5					AT %Q*	: BOOL;
	bOutputSpare6					AT %Q*	: BOOL;
	bOutputSpare7					AT %Q*	: BOOL;
	bOutputSpare8					AT %Q*	: BOOL;
	
	// nConcretePumpSpeed				AT %Q*	: INT;
	nDosingPumpSpeed				AT %Q*	: INT;
	nOutputSpare1					AT %Q*	: INT;
	nOutputSpare2					AT %Q*	: INT;
	
	
	//
	//Hardware RS-232
	stIn_EL6001 					AT %I*	: EL6inData22B;	
	stOut_EL6001 					AT %Q*	: EL6outData22B;
	
END_VAR

// ---- GVLs/GVLs/GVL_PN.TcGVL
{attribute 'qualified_only'}
// ***********************************************************************************
//
// Müller-steinag Gruppe, Kandergrien Einigen, CH-3646 Bern
// ETH Zurich, Building HIF E26, Laura-Hezner-Weg 7, CH-8093 Zürich
// 
// ***********************************************************************************
// 
// PROJECT     :  A061 Digital Casting System 
// FUNCTION    :  Global Profinet Varable input and output
// AUTHOR      :  Weiting Chen
// EMAIL       :  chenw@usi.ch
// Copyright   :  USI Mendrisio; ETH Zürich; Müller-steinag Gruppe (CH) 2023
//
// ***********************************************************************************

VAR_GLOBAL

	// Digital Output from robot (1 bit)
	DO_From_ROB AT %I* :ARRAY[0..31] OF BYTE; 
	// Group Output from robot (16 bit or 32 bit) 
	GO_From_ROB AT %I* :ARRAY[32..255] OF BYTE;
	// Digital Input to robot (1 bit)
	DI_To_ROB AT %Q* :ARRAY[0..31] OF arr8Bit;
	// Group Input to robot (16 bit or 32 bit)
	GI_To_ROB AT %Q* :ARRAY[32..255] OF BYTE;	

END_VAR

// ---- GVLs/GVLs/GVL_RESD.TcGVL
{attribute 'qualified_only'}
// ***********************************************************************************
//
// Müller-steinag Gruppe, Kandergrien Einigen, CH-3646 Bern
// ETH Zurich, Building Hin E26, Laura-Hezner-Weg 7, CH-8093 Zürich
// 
// ***********************************************************************************
// 
// PROJECT     :  A061 Digital Casting System 
// FUNCTION    :  Global Proninet Varable with robot
// AUTHOR      :  Weiting Chen
// EMAIL       :  chenw@usi.ch
// Copyright   :  USI Mendrisio; ETH Zürich; Müller-steinag Gruppe (CH) 2023
//
// **************S*********************************************************************

VAR_GLOBAL
	
CONCRETE_CONTROLLER: STRING := 'MIXER';//***********************************************************
b_Operate_mode_manual : BOOL;
b_Operate_mode_laptop : BOOL; 	
b_Operate_mode_robot : BOOL; 
b_Concrete_Controller_enable : BOOL;
b_Concrete_Controller_reset : BOOL;
b_Concrete_Controller_power_on : BOOL; 
n_Concrete_Controller_current_mode : INT;

MIXER: STRING := 'MIXER';//***********************************************************
// Inline Mixer
// input 		
b_MI1_set_run : BOOL;								// POWER ON *****
b_Ml1_Enable : BOOL;
n_MI1_set_speed : REAL;								// [0 rpm to 120 rpm]
b_MI1_set_curved_speed_mode_on: BOOL;				// Curved Speed Mode

// output 
b_MI1_Is_Run:BOOL;
b_MI1_Is_ready : BOOL;
n_MI1_status_SpeedM1 : INT;
n_MI1_status_SpeedM2 : INT;
f_Status_Torque_Motor_1 : REAL;
f_Status_Torque_Motor_2 : REAL;
f_MI1_status_temperature_funnel_outlet : REAL; 		
f_MI1_status_Pressure_funnel_inlet : REAL; 	
f_MI1_status_temperature_motor_1 : REAL; 			 
f_MI1_status_temperature_motor_2 : REAL; 
f_MI1_Override_Max_Speed : REAL := 120;				// [rpm]

CONCRETE_PUMP: STRING := 'CONCRETE_PUMP';
// Concrete Pump
// input
b_Concrete_Pump_Power_On: BOOL;						
b_Concrete_Pump_Forward_On: BOOL;					// Forward ON
b_Concrete_Pump_Backward_On: BOOL;					// X

b_Concrete_Pump_Flush_On: BOOL;						// FLUSH MODE ON 
n_Concrete_Pump_Flush_Flowrate: REAL;				// READ [l/min]

b_Concrete_Pump_Check_On: BOOL;						// CHECK MODE ON 
f_Concrete_Pump_Check_Flowrate: REAL; 				// [ O tp 24 l/min]
n_Concrete_Pump_Check_Duration: INT := 15; 			// [s]

f_Concrete_Pump_Set_Flowrate: REAL; 				// [0 to 24 l/min]
f_Concrete_Pump_dosing_volume: REAL := 0.32;		// calibrated 230926 WT
n_Concrete_Pump_Max_Speed : INT := 75;
n_Concrete_Pump_Set_Speed: INT;						// WRITE VALUE From 0 to 75 [rpm] 

b_CP1_is_run : BOOL;
b_CP1_is_ready : BOOL;
b_CP1_power_on :BOOL;
b_CP1_safety_grid_on : BOOL;
b_CP1_drive_error :BOOL;
f_CP1_status_temperature_concrete_fresh : REAL; // [°C]
f_CP1_status_temperature_Concrete_pump : REAL; // [°C] 
f_CP1_status_pressure_Concrete_pump: REAL; // [bar]


//f_Concrete_Pump_Density: REAL;					// [g/ml]
//f_Concrete_Pump_Check_Mass: REAL;           		// [g]

Admixture_Pump_1: STRING := 'Admixture Pump (AP1)';

b_Admixture_Pump_Power_On : BOOL;  					// Power On
b_Admixture_Pump_Set_Run : BOOL;  					// Set Run 
b_Admixture_Pump_Flush_On: BOOL;					// FLUSH MODE ON 
f_Admixture_Pump_Flush_Flowrate: REAL;				// READ 
b_Admixture_Pump_Check_On: BOOL;					// CHECK MODE ON 
f_Admixture_Pump_Check_Flowrate: REAL;				// READ 
n_Admixture_Pump_Check_Duration: INT := 60; 		// [s]
n_Admixture_Pump_Max_Flowrate :INT  := 606;		//calibrated 2402 WT
f_Admixture_Pump_Set_Flowrate: REAL;         		// 0 to 637 [ml/min] 
f_Admixture_Pump_dosing_factor: REAL := 1;			//only for scaled

//f_Admixture_Pump_1_Density: REAL;          // [g/ml]
//f_Admixture_Pump_1_Mass: REAL;             // [g]

b_Admixture_Pump_is_run : BOOL;
b_Admixture_Pump_is_ready : BOOL;
b_Admixture_Pump_no_error : BOOL;

//
Sup_Admixture_Pump_1: STRING := 'Admixture Pump (SP1)'; //***************************


b_Sup_Admixture_Pump_Power_On : BOOL;  					// Power On
b_Sup_Admixture_Pump_Set_Run: BOOL;  					// Set Run 

b_Sup_Admixture_Pump_Flush_On: BOOL;				// FLUSH MODE ON 
f_Sup_Admixture_Pump_Flush_Flowrate: REAL;
b_Sup_Admixture_Pump_Check_On: BOOL;				// CHECK MODE ON 
f_Sup_Admixture_Pump_Check_Flowrate: REAL;
n_Sup_Admixture_Pump_Check_Duration: INT := 60; 	// [s];
n_Sup_Admixture_Pump_Max_Flowrate:INT := 595; 		//[ml/min]

f_Sup_Admixture_Pump_Set_Flowrate: REAL;         	// 0 to 138[ml/min]
f_Sup_Admixture_Pump_dosing_factor:REAL:=1; //only for scaled

//f_Admixture_Pump_2_Density: REAL;          // [g/ml]
//f_Admixture_Pump_2_Mass: REAL;             // [g]

b_Sup_Admixture_Pump_is_run : BOOL;
b_Sup_Admixture_Pump_is_ready : BOOL;
b_Sup_Admixture_Pump_no_error : BOOL;
END_VAR

// ---- GVLs/GVLs/GVL_ROB.TcGVL
{attribute 'qualified_only'}
// ***********************************************************************************
//
// Müller-steinag Gruppe, Kandergrien Einigen, CH-3646 Bern
// ETH Zurich, Building Hin E26, Laura-Hezner-Weg 7, CH-8093 Zürich
// 
// ***********************************************************************************
// 
// PROJECT     :  A061 Digital Casting System 
// FUNCTION    :  Global Proninet Varable with robot
// AUTHOR      :  Weiting Chen
// EMAIL       :  chenw@usi.ch
// Copyright   :  USI Mendrisio; ETH Zürich; Müller-steinag Gruppe (CH) 2023
//
// **************S*********************************************************************

VAR_GLOBAL
	//output to robot digital input (DI) ; input from robot digital output(DO)
	
	//UINT type as 16bit ranged -32767 to 32767 (Here, the number is scaled by 1000
	
	//Concrete Controller
	ib_spare : BOOL;
	in_spare : INT;
	
	ib_CC1_enable : BOOL;
	ib_CC1_reset : BOOL;
	ib_CC1_data_recording : BOOL;
	
	ob_mode_manual : BOOL;
	ob_mode_laptop : BOOL; 	
	ob_mode_robot : BOOL; 
	on_current_mode : INT; //index use no scale.
	ob_CC1_power_on : BOOL; 
	
	//Inline Mixer (MI1)  				
	ib_MI1_set_run : BOOL;
	ib_MI1_enable : BOOL;
	ib_MI1_set_reset : BOOL;				 
	in_MI1_set_speed : UINT;								// [0 rpm to 120 rpm]
	ib_MI1_set_curved_speed_mode_on : BOOL;
	
	ob_MI1_is_run : BOOL;
	ob_MI1_is_ready : BOOL;
	
	on_MI1_status_speed_motor_1 : INT;				 	// [rpm]
	on_MI1_status_Speed_motor_2 : INT;					// [rpm]
	on_MI1_status_torque_motor_1 : REAL;					// [Nm]
	on_MI1_status_torque_motor_2 : REAL;					// [Nm]
	
	on_MI1_status_temperature_funnel_outlet : REAL; 		// [°C] 
	on_MI1_status_pressure_funnel_inlet : REAL; 			// [bar]
	on_MI1_status_temperature_motor_1 : REAL; 			// [°C] 
	on_MI1_status_temperature_motor_2 : REAL; 			// [°C] 
	
	
	//Concrete pump (CP1)  
	//ib_CP1_run: BOOL;					// NOT USE NOW
	ib_CP1_forward_on: BOOL;			    
	ib_CP1_backward_on: BOOL;			// 241219 Backward is not working from the conctroller
	in_CP1_set_flowrate: UINT; 			// 0 to 24 [l/min]
	in_CP1_set_speed: UINT;				// 0 to 75 [rpm] 
	in_CP1_set_dosing_volume: UINT;		// scale to 0 to 100 | calibration in 230926 WT 0.32
	
	ib_CP1_check_on: BOOL;			 
	in_CP1_set_check_Flowrate: UINT; 	// [l/min]
	t_CP1_set_check_duration: TIME;		//  T#1d2h30m40s500ms
	in_CP1_concrete_density: UINT;		// [g/ml]
	in_CP1_concrete_mass: UINT;          // [g]
	
	ib_CP1_flush_on: BOOL;				
	in_CP1_set_flush_flowrate: UINT;		// [l/min]
	
	on_CP1_status_temperature_concrete_fresh : REAL; // [°C]
	on_CP1_status_temperature_concrete_pump : REAL; // [°C] 
	on_CP1_status_pressure_concrete_pump: REAL; // [ bar
	
	ob_CP1_is_run : BOOL;
	ob_CP1_is_ready : BOOL;
	ob_CP1_power_on : BOOL;
	ob_CP1_safety_grid_on : BOOL;
	ob_CP1_drive_error :BOOL;
	

	
	
	// Admixture pump, High dosage ViscoTech Pump
	ib_AP1_power_on: BOOL; 
	ib_AP1_set_run: BOOL; 
	in_AP1_set_flowrate: UINT;         		// [ml/min] 
	in_AP1_set_dosing_factor: UINT;          // Set default 1
	
	ib_AP1_check_on: BOOL;			
	in_AP1_set_check_flowrate: UINT;
	t_AP1_set_check_duration: TIME;// T#1d2h30m40s500ms
	in_AP1_material_density: UINT;          // [g/ml]
	in_AP1_material_mass: UINT;             // [g]
	
	ib_AP1_flush_on: BOOL;			 
	in_AP1_set_flush_flowrate: UINT;	  // [ml/min] 
	
	ob_AP1_is_run : BOOL;
	ob_AP1_is_ready : BOOL;

	ob_AP1_no_error : BOOL;
	on_AP1_max_flowrate: UINT:=606;			// [ml/min] cailbrated 240710
	
	// Admixture pump, Low dosage ViscoTech Pump 
	ib_SP1_power_on: BOOL;
	ib_SP1_set_run: BOOL;
	in_SP1_set_flowrate: UINT;         // [ml/min]
	in_SP1_dosing_factor:UINT;       
	
	ib_SP1_set_check_on: BOOL;			 
	in_SP1_set_check_flowrate: UINT;	  // [ml/min] 
	t_SP1_Check_Duration: TIME ;       // T#1d2h30m40s500ms
	in_SP1_material_density: UINT;     // [g/ml]
	in_SP1_material_mass: UINT;        // [g]
	
	ib_SP1_flush_on: BOOL;			 
	in_SP1_flush_flowrate: UINT;		// [ml/min] 
	
	ob_SP1_is_run:BOOL;
	ob_SP1_is_ready : BOOL;
	ob_SP1_no_error : BOOL;
	on_SP1_max_flowrate:UINT := 148;	 // [ml/min] cailbrated 240710
	
END_VAR

// ---- GVLs/GVLs/ReadMe.TcGVL
{attribute 'qualified_only'}
// ***********************************************************************************
//
// Müller-steinag Gruppe, Kandergrien Einigen, CH-3646 Bern
// ETH Zurich, Building HIF E26, Laura-Hezner-Weg 7, CH-8093 Zürich
// 
// ***********************************************************************************
// 
// PROJECT     :  A061 Digital Casting System 
// FUNCTION    :  Profinet Variable Convertor
// AUTHOR      :  Weiting Chen
// EMAIL       :  chenw@usi.ch
// Copyright   :  USI Mendrisio; ETH Zürich; Müller-steinag Gruppe (CH) 2023
// Contributor :  Fabio Scotto / Philippe Fleischmann 
//
// ***********************************************************************************

VAR_GLOBAL
	
(*
Set the IP with 192.168.30.11 


File description 
GVL(GVL : Global variables)
GVL_IO(GVL_IO : IO)
GVL_PN(GVL_PN : Profinet Array)
GVL_RED(GVL_research : variables for control via laptop)
GVL_ROB(GVL_research : variables for control via Robot)


Data Type Prefix
ib = Input Bool   / ob = Output Bool
if = Input float  / of = Output float (REAL, LREAL)
in = Input numeric/ on = Output numeric 
(INT, SINT, USINT, UNIT, DINT, UDINT, BYTE, WORD, DWORD, LWORD, XINT, UXINT, XWORD) 
t = Time (TON)
s = String


Naming Shortcuts
CC1 = Concrete Controller 
AP1 = Admixture pump, High dosage ViscoTech Pump (Xseed or Accelerator)
CP1 = Concrete Pump
SP1 = Admixture pump, Low dosage ViscoTech Pump  (Xseed or Accelerator or Superplasticizer)

PP1 = Peristaltic Pump
MI1 = Mixer
RED = Research Data
PN = Profinet with Roboter

*)

END_VAR

// ---- POUs/MAIN.TcPOU
PROGRAM MAIN
VAR

END_VAR

// ***********************************************************************************
//
// Müller-steinag Gruppe, Kandergrien Einigen, CH-3646 Bern
// ETH Zurich, Building HIF E26, Laura-Hezner-Weg 7, CH-8093 Zürich
// 
// ***********************************************************************************
// 
// PROJECT     :  A061 Digital Casting System 
// FUNCTION    :  Main 
// AUTHOR      :  Weiting Chen
// EMAIL       :  chenw@usi.ch
// Copyright   :  USI Mendrisio; ETH Zürich; Müller-steinag Gruppe (CH) 2024
//
// ***********************************************************************************


P_Control_Mode();

// data comunicaiton robot via EL6631

IF GVL.b_mode_laptop THEN 
	P_Laptop_Operate();
ELSIF GVL.b_mode_robot THEN 
	P_PNDataConvert();
	P_Robot_Operate();
ELSIF GVL.b_mode_manual THEN 
	P_Manual_Operate();
END_IF


// ELSE
// 	temp_speed_override:=F_ScalAnalogOut(
// 		n_Input:= REAL_TO_INT(GVL_IO.in_MI1_Poti_Speed),
// 		n_InMin:= 0,
// 		n_InMax:= 32767,
// 		n_OutMin:= 0,
// 		n_OutMax:= 100);
// END_IF

// GVL_VAR.f_MI1_Override:= temp_speed_override;

END_PROGRAM

// ---- POUs/P_Control_Mode.TcPOU
PROGRAM P_Control_Mode
VAR
END_VAR

// ***********************************************************************************
//
// Müller-steinag Gruppe, Kandergrien Einigen, CH-3646 Bern
// ETH Zurich, Building HIF E26, Laura-Hezner-Weg 7, CH-8093 Zürich
// 
// ***********************************************************************************
// 
// PROJECT     :  A061 Digital Casting System 
// FUNCTION    :  Control mode 
// AUTHOR      :  Weiting Chen
// EMAIL       :  chenw@usi.ch
// Copyright   :  USI Mendrisio; ETH Zürich; Müller-steinag Gruppe (CH) 2023
//
// ***********************************************************************************

GVL.b_mode_manual := GVL_IO.ib_CC1_Button_Mode_Manual; 
GVL.b_mode_laptop := GVL_IO.ib_CC1_Button_Mode_Laptop;


GVL.b_mode_robot := False;
IF GVL.b_mode_manual THEN 
	GVL.s_current_mode := 'Controller';
ELSIF GVL.b_mode_laptop  THEN
	GVL.s_current_mode := 'Laptop';
ELSIF NOT GVL.b_mode_manual AND NOT GVL.b_mode_laptop THEN
	GVL.s_current_mode := 'Robot';
	GVL.b_mode_robot := TRUE;
ELSE
	GVL.s_current_mode := 'None';
END_IF

END_PROGRAM

// ---- POUs/P_Laptop_Operate.TcPOU
PROGRAM P_Laptop_Operate
VAR
	fb_MC_SetPosition : FB_SoEAX5000SetPositionOffset;
	pos:LREAL;
	Mixer1_2		: FB_Mixer1_2;
	Analog			: FB_Analog;
	SafetyReset 	: bool;
	b_Enable		: BOOL;
	b_Reset			: BOOL;
	
	Test : MC_ReadStatus;
	
	speed : REAL;
	fb_SetOutputDataToIO : FB_SetOutputDataToIO;
	fb_getOutputData : FB_GetOutputData;
	fb_setConfig : FB_SetConfigData;
	
	//
	b_Safety_Reset : BOOL;
	b_Timer_Rest : BOOL;
	t_CC1_Time_Safety_Rest : TIME :=T#5S; //wait 5s for controller restart
	fb_CC1_Trigger_Safety_On : R_TRIG;
	fb_CC1_Trigger_Safety_Off : R_TRIG;
	fb_CC1_Timer_Safety: TON;

END_VAR

// ***********************************************************************************
//
// Müller-steinag Gruppe, Kandergrien Einigen, CH-3646 Bern
// ETH Zurich, Building HIF E26, Laura-Hezner-Weg 7, CH-8093 Zürich
// 
// ***********************************************************************************
// 
// PROJECT     :  A061 Digital Casting System 
// FUNCTION    :  Laptop operate process
// AUTHOR      :  Weiting Chen
// EMAIL       :  chenw@usi.ch
// Copyright   :  USI Mendrisio; ETH Zürich; Müller-steinag Gruppe (CH) 2024
//
// ***********************************************************************************


b_Timer_Rest:=GVL_RESD.b_Concrete_Controller_reset;

//controller reset trigger
fb_CC1_Timer_Safety(
					IN:=b_Timer_Rest,
					PT:=t_CC1_Time_Safety_Rest);

fb_CC1_Trigger_Safety_On(clk:=fb_CC1_Timer_Safety.IN);
fb_CC1_Trigger_Safety_Off(clk:=fb_CC1_Timer_Safety.Q);
//b_Safety_Reset:=FALSE;
IF fb_CC1_Trigger_Safety_On.Q THEN
	b_Safety_Reset:=TRUE;
END_IF
IF fb_CC1_Trigger_Safety_Off.Q THEN 
	b_Safety_Reset:=FALSE;
	GVL_RESD.b_Concrete_Controller_reset:=FALSE;
END_IF
GVL_IO.ob_CC1_Safety_Reset:= b_Safety_Reset OR GVL_IO.ib_CC1_Button_Reset;

// Concrete Conctroller enable 
P_CC1_Enable( b_set_run:= GVL_RESD.b_Concrete_Controller_enable );



//***********************************************************************************
// Set Process Configuration
//***********************************************************************************

fb_setConfig(
// Gerenal
// Concrete Controller
// Inline Mixer
_f_MI1_Override_Max_Speed :=120,

// Concrete Pump
_f_CP1_Max_Flowrate := INT_TO_REAL(GVL_RESD.n_Concrete_Pump_Max_Speed) * 
								   GVL_RESD.f_Concrete_Pump_dosing_volume,
_f_CP1_Check_Flowrate := GVL_RESD.f_Concrete_Pump_Check_Flowrate,
_t_CP1_Check_Duration := INT_TO_TIME(GVL_RESD.n_Concrete_Pump_Check_Duration)*1000,

// Admixture pump (High)
_n_AP1_Max_Flowrate := GVL_RESD.n_Admixture_Pump_Max_Flowrate,
_n_AP1_Check_Flowrate := GVL_RESD.f_Admixture_Pump_Check_Flowrate,
_t_AP1_Check_Duration := INT_TO_TIME(GVL_RESD.n_Admixture_Pump_Check_Duration)*1000,
_n_AP1_Flush_Flowrate := GVL_RESD.f_Admixture_Pump_Flush_Flowrate,
//_f_AP1_Check_Mass : REAL;

// Admixture pump (low)
_n_SP1_Max_Flowrate := GVL_RESD.n_Sup_Admixture_Pump_Max_Flowrate,
_n_SP1_Check_Flowrate := GVL_RESD.f_Sup_Admixture_Pump_Check_Flowrate,
_t_SP1_Check_Duration := INT_TO_TIME(GVL_RESD.n_Sup_Admixture_Pump_Check_Duration)*1000,
//_f_SP1_Check_Mass : REAL;
);

//***********************************************************************************
// Setup IO data to PLC
//***********************************************************************************	
fb_SetOutputDataToIO(		
	// Mixer 
	b_MI1_set_run := GVL_RESD.b_MI1_set_run,
	b_Ml1_Enable := GVL_RESD.b_Ml1_Enable,
	b_MI1_Curved_Speed_On := GVL_RESD.b_MI1_set_curved_speed_mode_on,
	f_MI1_Override_Speed := GVL_RESD.n_MI1_set_speed,
	f_MI1_Override_Max_Speed := GVL_RESD.f_MI1_Override_Max_Speed,
	
	// Concrete Pump
	b_CP1_Forward_On := GVL_RESD.b_Concrete_Pump_Forward_On,
	b_CP1_Backward_On := GVL_RESD.b_Concrete_Pump_Backward_On,
	b_CP1_Flush_On := GVL_RESD.b_Concrete_Pump_Flush_On,
	b_CP1_Check_On := GVL_RESD.b_Concrete_Pump_Check_On,
	n_CP_Flowrate_mode := TRUE,
	n_CP1_Operate_Flowrate := REAL_TO_UDINT(GVL_RESD.f_Concrete_Pump_Set_Flowrate*100),
	n_CP1_Check_Flowrate := REAL_TO_UDINT(GVL_RESD.f_Concrete_Pump_Check_Flowrate*100),
	n_CP1_Flush_Flowrate := REAL_TO_UDINT(GVL_RESD.n_Concrete_Pump_Flush_Flowrate*100),
	f_dosing_volume := REAL_TO_INT(GVL_RESD.f_Concrete_Pump_dosing_volume*100),
	
	n_CP1_max_speed := GVL_RESD.n_Concrete_Pump_Max_Speed,
	n_CP1_target_speed := GVL_RESD.n_Concrete_Pump_Set_Speed,

	// Admixture pump (High)
	b_AP1_Power_On := GVL_RESD.b_Admixture_Pump_Power_On,
	b_AP1_Run := GVL_RESD.b_Admixture_Pump_Set_Run,
	b_AP1_Flush_On := GVL_RESD.b_Admixture_Pump_Flush_On,
	b_AP1_Check_On := GVL_RESD.b_Admixture_Pump_Check_On,
	
	n_AP1_Flowrate_mode := TRUE,
	n_AP1_Max_Flowrate := GVL_RESD.n_Admixture_Pump_Max_Flowrate,
	n_AP1_Operate_Flowrate := REAL_TO_UDINT(GVL_RESD.f_Admixture_Pump_Set_Flowrate*10),
	n_AP1_Check_Flowrate := REAL_TO_UDINT(GVL_RESD.f_Admixture_Pump_Check_Flowrate*10),
	n_AP1_Flush_Flowrate := REAL_TO_UDINT(GVL_RESD.f_Admixture_Pump_Flush_Flowrate*10),
	n_AP1_Dosing_factor := REAL_TO_INT(GVL_RESD.f_Admixture_Pump_dosing_factor*10),
	
	// Admixture pump (High)
	b_SP1_Power_On := GVL_RESD.b_Sup_Admixture_Pump_Power_On,
	b_SP1_Run := GVL_RESD.b_Sup_Admixture_Pump_Set_Run,
	b_SP1_Flush_On := GVL_RESD.b_Sup_Admixture_Pump_Flush_On,
	b_SP1_Check_On := GVL_RESD.b_Sup_Admixture_Pump_Check_On,
	
	n_SP1_Flowrate_mode := TRUE,
	n_SP1_Max_Flowrate := GVL_RESD.n_Sup_Admixture_Pump_Max_Flowrate,
	n_SP1_Operate_Flowrate := REAL_TO_UDINT(GVL_RESD.f_Sup_Admixture_Pump_Set_Flowrate*10),
	n_SP1_Check_Flowrate := REAL_TO_UDINT(GVL_RESD.f_Sup_Admixture_Pump_Check_Flowrate*10),
	n_SP1_Flush_Flowrate := REAL_TO_UDINT(GVL_RESD.f_Sup_Admixture_Pump_Flush_Flowrate*10),
	n_SP1_Dosing_factor := REAL_TO_INT(GVL_RESD.f_Sup_Admixture_Pump_dosing_factor*10),
	);

//***********************************************************************************
// Inline Mixer
//***********************************************************************************
	//mixer 
Mixer1_2(
	Mixer1			:= GVL.Axis_Mixer1,
	Mixer2			:= GVL.Axis_Mixer2,
	f_Velocity		:= GVL.f_MI1_MaxSpeed,
	b_JogForward	:= FALSE,
	b_JogBackwards	:= fb_SetOutputDataToIO.b_MI1_set_run,
	b_Enable		:= fb_SetOutputDataToIO.b_Ml1_Enable AND GVL_IO.ib_CC1_Safety_Ready,
	b_Reset			:= GVL_RESD.b_Concrete_Controller_reset OR GVL_IO.ib_CC1_Button_Reset,
	f_Override		:= GVL.n_MI1_OverrideSpeed,
	);
	(*
	fb_MC_SetPosition(
	Axis			:= GVL.Axis_Mixer2,
	memory			:= 1,
	Feedback		:= 0);*)
pos:=GVL.Axis_Mixer2.NcToPlc.ModuloActPos;
GVL.b_MI1_ReadToDrive:=Mixer1_2.b_ReadyToDrive;
P_MI1_OnOff(b_set_run := fb_SetOutputDataToIO.b_MI1_set_run,);

//***********************************************************************************
// Concrete Pump
//***********************************************************************************

// concrete pump power control is from pump itself
P_CP1_Enable();
P_CP1_Check(b_set_run := fb_SetOutputDataToIO.b_CP1_Forward_On,
			b_check_mode_on := fb_SetOutputDataToIO.b_CP1_Check_On,
			t_check_duration := fb_setConfig._t_CP1_Check_Duration,
			);


//***********************************************************************************
// Acceleration Pump
//***********************************************************************************

// Acceleration Pump 1 check
P_AP1_Check(b_set_run := fb_SetOutputDataToIO.b_AP1_Run,
			b_check_mode_on := fb_SetOutputDataToIO.b_AP1_Check_On,
			t_check_duration := fb_setConfig._t_AP1_Check_Duration,
			);
// Check for Acceleration Pump 1 state
IF NOT fb_SetOutputDataToIO.b_AP1_Check_On THEN
//
// Acceleration Pump 1 On/Off
	P_AP1_OnOff(b_set_run := fb_SetOutputDataToIO.b_AP1_Run);
END_IF

//***********************************************************************************
// Superplasticizer Pump
//***********************************************************************************

// Superplasticizer Pump 1 Check (220916 WT
P_SP1_Check(b_set_run := fb_SetOutputDataToIO.b_SP1_Run,
			b_check_mode_on := fb_SetOutputDataToIO.b_SP1_Check_On,
			t_check_duration := fb_setConfig._t_SP1_Check_Duration,
			);
IF NOT fb_SetOutputDataToIO.b_SP1_Check_On THEN
	P_SP1_OnOff(b_set_run := fb_SetOutputDataToIO.b_SP1_Run);
END_IF

//***********************************************************************************
// Get out put data from PLC
//***********************************************************************************
fb_getOutputData(
	
	//CC1
	b_mode_manual := GVL_RESD.b_Operate_mode_manual,
	b_mode_laptop := GVL_RESD.b_Operate_mode_laptop, 	
	b_mode_robot := GVL_RESD.b_Operate_mode_robot, 
	b_CC1_power_on := GVL_RESD.b_Concrete_Controller_power_on, 
	n_current_mode := GVL_RESD.n_Concrete_Controller_current_mode,

	//MI1
	b_MI1_Is_Run := GVL_RESD.b_MI1_Is_Run,
	b_MI1_is_ready := GVL_RESD.b_MI1_Is_Ready,
	n_MI1_status_SpeedM1 := GVL_RESD.n_MI1_status_SpeedM1,
	n_MI1_status_SpeedM2 := GVL_RESD.n_MI1_status_SpeedM2,
	f_Status_Torque_Motor_1 := GVL_RESD.f_Status_Torque_Motor_1,
	f_Status_Torque_Motor_2 := GVL_RESD.f_Status_Torque_Motor_2,
	f_MI1_status_temperature_funnel_outlet := GVL_RESD.f_MI1_status_temperature_funnel_outlet, 		
	f_MI1_status_Pressure_funnel_inlet := GVL_RESD.f_MI1_status_Pressure_funnel_inlet, 	
	f_MI1_status_temperature_motor_1  := GVL_RESD.f_MI1_status_temperature_motor_1, 			 
	f_MI1_status_temperature_motor_2  := GVL_RESD.f_MI1_status_temperature_motor_2,

	//CP1
	b_CP1_is_run := GVL_RESD.b_CP1_is_run,
	b_CP1_is_ready := GVL_RESD.b_CP1_is_ready,
	
	b_CP1_is_ready := GVL_ROB.ob_CP1_is_ready,
	b_CP1_power_on := GVL_ROB.ob_CP1_power_on,
	b_CP1_safety_grid_on := GVL_ROB.ob_CP1_safety_grid_on,
	b_CP1_drive_error := GVL_ROB.ob_CP1_drive_error,
	
	f_CP1_status_temperature_concrete_fresh := GVL_RESD.f_CP1_status_temperature_concrete_fresh,
	f_CP1_status_temperature_Concrete_pump := GVL_RESD.f_CP1_status_temperature_Concrete_pump,
	f_CP1_status_pressure_Concrete_pump := GVL_RESD.f_CP1_status_pressure_Concrete_pump,
	
	//AP1
	b_AP1_is_run := GVL_RESD.b_Admixture_Pump_is_run,
	b_AP1_is_ready := GVL_RESD.b_Admixture_Pump_is_ready,
	b_AP1_no_error := GVL_RESD.b_Admixture_Pump_no_error,
	
	//SP1
	b_SP1_is_run := GVL_RESD.b_Sup_Admixture_Pump_is_run,
	b_SP1_is_ready := GVL_RESD.b_Sup_Admixture_Pump_is_ready,
	b_SP1_no_error := GVL_RESD.b_Sup_Admixture_Pump_no_error,
);

END_PROGRAM

// ---- POUs/Component/MIxer_Driver/FB_Mixer1_2.TcPOU
FUNCTION_BLOCK FB_Mixer1_2
VAR_INPUT
	// General
	b_Enable				: BOOL;		
	b_Reset					: BOOL;
	
	// Parameter SetPosition
	b_ModeSetPosition		: BOOL;				// Active Mode SetPosition
	b_SetPositionMixer1		: BOOL;				// SetPositon mixer 1 with f_SetPosition1
	b_SetPositionMixer2		: BOOL;				// SetPositon mixer 2 with f_SetPosition1
	f_SetPositionMixer1		: LREAL;			
	f_SetPositionMixer2		: LREAL;			
	
	//Parameter positions
	f_OffsetPositionMixer1 	: LREAL;			// 0..360°
	f_OffsetPositionMixer2 	: LREAL;			// 0..360°	
	f_CollisionPosMin		: LREAL := 35; 		// 0°..f_CollisionPosMax
	f_CollisionPosMax		: LREAL	:= 145;		// f_CollisionPosMin..180°
	f_OffsetMixer1Mixer2	: LREAL := 90; 		//0..360°
	
	//
	// Parameter drive
	f_Override				: LREAL;
	f_Velocity				: LREAL;
	b_JogForward			: BOOL;
	b_JogBackwards			: BOOL;
END_VAR
VAR_OUTPUT
	b_PowerActiveMixer1		: BOOL;
	b_PowerActiveMixer2		: BOOL;
	b_ReadyToDrive			: BOOL;
	b_ErrorGen				: BOOL;
	b_ErrorMixer1			: BOOL;
	b_ErrorMixer2			: BOOL;
	n_ErrorIDMixer1			: UDINT;
	n_ErrorIDMixer2			: UDINT;
	f_ActVelocityMixer1		: LREAL;
	f_ActVelocityMixer2		: LREAL;
	f_ActTorqueMixer1		: LREAL;
	f_ActTorqueMixer2		: LREAL;
	f_ActPositionMixer1		: LREAL;
	f_ActPositionMixer2		: LREAL;
END_VAR
VAR_IN_OUT
	Mixer1					: AXIS_REF;
	Mixer2					: AXIS_REF;
END_VAR
VAR		
	n_Step					: INT;				// Step chain
	b_ErrorInt				: BOOL;				// Error Intern

	b_Mixer1InCollision		: BOOL;				// Check if paddle mixer 1 in collision zone
	b_Mixer2InCollision		: BOOL;				// Check if paddle mixer 2 in collision zone
	f_PositionMixer1		: LREAL; 			// Position paddle mixer 1 in 0°..180°
	f_PositionMixer2		: LREAL; 			// Position paddle mixer 2 in 180°..360° (scaled 180°..0°)                                               
	f_ActPositionMixer1Calc	: LREAL;			// Actual position mixer 1 (with offset)
	f_ActPositionMixer2Calc	: LREAL;			// Actual position mixer 2 (with offset)

	// FBs	
	fb_Mixer1				: FB_Drive;	
	fb_Mixer2				: FB_Drive;	
	fb_MC_GearIn			: MC_GearIn;
	fb_MC_GearOut			: MC_GearOut;	
	fb_MC_ReadStatusMixer1	: MC_ReadStatus;
	fb_MC_ReadStatusMixer2	: MC_ReadStatus;
END_VAR

//***********************************************************************************
//
// ETH Zürich / Robotic Fabrication Lab
// HIB C 13 / Stefano-Franscini-Platz 1
// CH-8093 Zürich
// 
// ***********************************************************************************
// 
// PROJECT     :  ?? 
// 
// FUNCTION    :  FB_DriveGea
// 
// AUTHOR      :  Mathias Suter
// 
// EMAIL       :  mathias.suter@solinaut.ch
// 
// Copyright   :  ETH Zürich (CH) 2021
//
// ***********************************************************************************

//
// Limit f_OffsetPositionMixer1 and f_OffsetPositionMixer2 to 0°..360°
IF f_OffsetPositionMixer1 < 0 THEN
	f_OffsetPositionMixer1 := 0;
END_IF
IF f_OffsetPositionMixer1 > 360 THEN
	f_OffsetPositionMixer1 := 360;
END_IF

IF f_OffsetPositionMixer2 < 0 THEN
	f_OffsetPositionMixer2 := 0;
END_IF
IF f_OffsetPositionMixer2 > 360 THEN
	f_OffsetPositionMixer2 := 360;
END_IF

//
// Calculate and limit f_ActPosition1Calc and f_ActPosition1Calc to 0°..360°
f_ActPositionMixer1Calc := f_ActPositionMixer1 + f_OffsetPositionMixer1;
IF f_ActPositionMixer1Calc < 0 THEN
	f_ActPositionMixer1Calc := f_ActPositionMixer1Calc + 360;
ELSIF f_ActPositionMixer1Calc > 360 THEN
	f_ActPositionMixer1Calc := f_ActPositionMixer1Calc - 360;
END_IF

f_ActPositionMixer2Calc := f_ActPositionMixer2 + f_OffsetPositionMixer2;
IF f_ActPositionMixer2Calc < 0 THEN
	f_ActPositionMixer2Calc := f_ActPositionMixer1Calc + 360;
ELSIF f_ActPositionMixer2Calc > 360 THEN
	f_ActPositionMixer2Calc := f_ActPositionMixer1Calc - 360;
END_IF

//
// Calculate which position has the mixer 1 paddle in 0°-180° zone (f_ActPosition1Calc or f_ActPosition1Calc + 180°)
// for checking collision
IF f_ActPositionMixer1Calc < 180 THEN
	f_PositionMixer1 := f_ActPositionMixer1Calc;
ELSE	
	f_PositionMixer1 := f_ActPositionMixer1Calc - 180;
END_IF

//
// Calculate which position has the mixer 1 paddle in 180°-360° zone (f_ActPosition2Calc or f_ActPosition2Calc + 180°) 
// scale position 180° - 360° to 180° - 0°, for checking collision
(*IF f_ActPositionMixer2Calc < 180 THEN
	f_PositionMixer2 := 180 - f_ActPositionMixer2Calc;
ELSE	
	f_PositionMixer2 := 360 - f_ActPositionMixer2Calc;
END_IF*)

IF f_ActPositionMixer2Calc < 180 THEN
	f_PositionMixer2 := f_ActPositionMixer2Calc;
ELSE	
	f_PositionMixer2 := f_ActPositionMixer2Calc - 180;
END_IF

//
//Check if paddle in collision zone
b_Mixer1InCollision := f_PositionMixer1 > f_CollisionPosMin AND f_PositionMixer1 < f_CollisionPosMax;
b_Mixer2InCollision := f_PositionMixer2 > f_CollisionPosMin AND f_PositionMixer2 < f_CollisionPosMax;

//
// Limit offset mixer 1 to mixer 2 (for driving)
IF f_OffsetMixer1Mixer2 < 0 THEN
	f_OffsetMixer1Mixer2 := 0;
END_IF
IF f_OffsetMixer1Mixer2 > 360 THEN
	f_OffsetMixer1Mixer2 := 360;
END_IF

fb_MC_ReadStatusMixer1(Axis:=Mixer1,
					Enable:=TRUE);

fb_MC_ReadStatusMixer2(Axis:=Mixer2,
					Enable:=TRUE);


//
// Step chain for Gear In two Axis
CASE n_step OF
	
	0:
		//
		// Init
		n_Step := 10;
	
	10:
		//
		// Enable or set position
		IF b_Enable THEN
			n_Step := 20;
		END_IF;
		
		//
		// Error
		IF b_ErrorInt THEN
			n_Step := 200;
		END_IF
			
	20:
		//
		// GearOut
		IF fb_MC_GearOut.Done THEN
			n_Step := 30;
		END_IF
		
		//
		// Not Enable or Error	
		IF NOT b_Enable THEN
			n_Step := 10;
 		ELSIF b_ErrorInt THEN
			n_Step := 200;
		END_IF

	30:
		//
		//Set position posible (via b_SetPosition1 or b_SetPosition2 to value f_SetPosition1/f_SetPosition2)
				
		//
		// End set position 
		IF NOT b_ModeSetPosition THEN
			n_Step := 35;
		END_IF
			
		//
		// Not Enable or Error	
		IF NOT b_Enable THEN
			n_Step := 10;
 		ELSIF b_ErrorInt THEN
			n_Step := 200;
		END_IF
	35:
		//
		//Enable
		IF fb_Mixer1.b_PowerActive AND fb_Mixer2.b_PowerActive THEN
			n_Step := 40;	
		END_IF
		
		//
		// Not Enable or Error	
		IF NOT b_Enable THEN
			n_Step := 10;
 		ELSIF b_ErrorInt THEN
			n_Step := 200;
		END_IF
		
	40:
		//
		// Check mixer 1 or mixer 2 in collision zone
		IF b_Mixer1InCollision OR b_Mixer1InCollision THEN
			IF f_PositionMixer1 < f_PositionMixer2 THEN 
				//
				// Drive backwards out off collision zone
				n_Step := 50;
			ELSE
				//
				// Drive forward  out off collision zone
				n_Step := 60;
			END_IF;
		ELSE
			//
			// No driving
			n_Step := 70;
		END_IF
		
		//
		// Not Enable or Error	
		IF NOT b_Enable THEN
			n_Step := 10;
 		ELSIF b_ErrorInt THEN
			n_Step := 200;
		END_IF
		
	50:
		//
		// Drive till mixer 1 and mixer 2 not in collision zone (drive backwards)
		IF NOT b_Mixer1InCollision AND NOT b_Mixer2InCollision THEN
			n_Step := 70;
		END_IF
				
		//
		// Not Enable or Error	
		IF NOT b_Enable THEN
			n_Step := 10;
 		ELSIF b_ErrorInt THEN
			n_Step := 200;
		END_IF

	60:
		//
		// Drive till mixer 1 and mixer 2 not in collision zone (drive forward)
		IF NOT b_Mixer1InCollision AND NOT b_Mixer2InCollision THEN
			n_Step := 70;
		END_IF
		
		//
		// Not Enable or Error	
		IF NOT b_Enable THEN
			n_Step := 10;
 		ELSIF b_ErrorInt THEN
			n_Step := 200;
		END_IF
					
	70:
		//
		// Check mixer 1 and mixer 2 standstill
		IF Mixer1.Status.StandStill AND Mixer2.Status.StandStill THEN
			//
			// Calculate offset mixer 1 to mixer 2
			IF (f_ActPositionMixer1Calc + f_OffsetMixer1Mixer2) > 360 THEN
				fb_Mixer2.f_Position := f_ActPositionMixer1Calc + f_OffsetMixer1Mixer2 - 360;
			ELSE	
				fb_Mixer2.f_Position := f_ActPositionMixer1Calc + f_OffsetMixer1Mixer2;
			END_IF
			
			n_Step := 80;		
		END_IF
	
		//
		// Not Enable or Error	
		IF NOT b_Enable THEN
			n_Step := 10;
 		ELSIF b_ErrorInt THEN
			n_Step := 200;
		END_IF

	80:
		//
		//
		n_Step := 85;
		
		//
		// Not Enable or Error	
		IF NOT b_Enable THEN
			n_Step := 10;
 		ELSIF b_ErrorInt THEN
			n_Step := 200;
		END_IF
		
	85:
		//
		//
		IF fb_Mixer2.b_MoveAbsoluteDone THEN
			n_Step := 100;
		END_IF		
			
		//
		// Not Enable or Error	
		IF NOT b_Enable THEN
			n_Step := 10;
 		ELSIF b_ErrorInt THEN
			n_Step := 200;
		END_IF

	100:
		//
		// Couple
		IF fb_MC_GearIn.InGear THEN
			n_Step := 110;
		END_IF;
		
		//
		// Not Enable or Error
		IF NOT b_Enable THEN
			n_Step := 10;
 		ELSIF b_ErrorInt THEN
			n_Step := 200;
		END_IF	
	
	110:
		//
		//  Jog command possible (Coupled) via b_JogForward/b_JogBackwards
		
		
		//
		// Go to mode set position
		IF b_ModeSetPosition THEN
			n_Step := 20;	
		END_IF
		
		//
		// Not Enable or Error
		IF NOT b_Enable THEN
			n_Step := 10;
 		ELSIF b_ErrorInt THEN
			n_Step := 200;
		END_IF		
						
	200:
		// 	
		// GearOut
		IF fb_MC_GearOut.Done THEN
			n_Step := 210;
		END_IF
	
	210:
		//
		// No Error		
		IF NOT b_ErrorInt AND (b_Reset or not b_Enable) THEN
			n_Step := 10;
		END_IF
		
END_CASE


//
// Errors
b_ErrorInt:= fb_Mixer1.b_Error OR fb_Mixer2.b_Error OR fb_MC_GearIn.Error OR fb_MC_GearOut.Error;

IF b_reset THEN
	fb_MC_GearOut.Execute:=FALSE;
	fb_MC_GearIn.Execute:=FALSE;
END_IF

//
// Outputs
b_PowerActiveMixer1			:= fb_Mixer1.b_PowerActive;
b_PowerActiveMixer2			:= fb_Mixer2.b_PowerActive;
b_ReadyToDrive				:= n_Step = 110;
b_ErrorGen					:= b_ErrorInt;
b_ErrorMixer1				:= fb_Mixer1.b_Error;
b_ErrorMixer2				:= fb_Mixer2.b_Error;
n_ErrorIDMixer1				:= fb_Mixer1.n_ErrorID;
n_ErrorIDMixer2				:= fb_Mixer2.n_ErrorID;
f_ActVelocityMixer1			:= fb_Mixer1.f_ActVelocity;
f_ActVelocityMixer2			:= fb_Mixer2.f_ActVelocity;
f_ActTorqueMixer1			:= fb_Mixer1.f_ActTorque;
f_ActTorqueMixer2			:= fb_Mixer2.f_ActTorque;
f_ActPositionMixer1			:= fb_Mixer1.f_ActPosition;
f_ActPositionMixer2			:= fb_Mixer2.f_ActPosition;
	
 
//
// Set position for mode SetPosition
IF n_Step = 30 THEN
	fb_Mixer1.f_Position := f_SetPositionMixer1;		
	fb_Mixer2.f_Position := f_SetPositionMixer2;
END_IF

//		
// Set velocity for Mixer 1/2		
IF n_Step = 110 THEN  
	fb_Mixer1.f_Velocity := f_Velocity;		   
	fb_Mixer2.f_Velocity := f_Velocity;	
ELSE
	fb_Mixer1.f_Velocity := 10;		   
	fb_Mixer2.f_Velocity := 10;
	f_Override:=100;
END_IF	   

//
// FB Mixer1
fb_Mixer1(
	Axis 					:= Mixer1,
	b_Enable 				:= b_Enable AND n_Step >= 35 AND n_Step <= 110,
	b_Reset					:= b_Reset AND NOT b_Enable,
	b_JogForward			:= (n_Step = 60 AND b_Mixer1InCollision) OR (n_Step = 110 AND b_JogForward),	  
	b_JogBackwards			:= (n_Step = 50 AND b_Mixer1InCollision) OR (n_Step = 110 AND b_JogBackwards),	
	b_MoveAbsolute			:= FALSE,
	n_MoveAbsoluteDirection := MC_Shortest_Way,
	b_Home					:= n_Step = 30 AND b_SetPositionMixer1,
	f_Acceleration			:= 0,
	f_Deceleration			:= 0,	
	f_Jerk					:= 0,
	f_Override 				:= f_Override);

	
//
// FB Mixer2
fb_Mixer2(
	Axis 					:= Mixer2,
	b_Enable 				:= b_Enable AND n_Step >= 35 AND n_Step <= 110,
	b_Reset					:= b_Reset AND NOT b_Enable,
	b_JogForward			:= (n_Step = 50 AND b_Mixer2InCollision),  
	b_JogBackwards			:= (n_Step = 60 AND b_Mixer2InCollision),	
	b_MoveAbsolute			:= n_Step = 80 OR n_Step = 85,
	n_MoveAbsoluteDirection := MC_Shortest_Way,
	b_Home					:= n_Step = 30 AND b_SetPositionMixer2,
	f_Acceleration			:= 0,
	f_Deceleration			:= 0,	
	f_Jerk					:= 0,
	f_Override 				:= f_Override);

//
// FB GearIn	
fb_MC_GearIn(
	Master 					:= Mixer1,
	Slave					:= Mixer2,
	Execute					:= b_Enable AND (n_Step = 100),
	RatioNumerator 			:= 1,
	RatioDenominator 		:= 1);
	                    	
//                      	
// FB GearOut           	
fb_MC_GearOut(          	
	Slave 					:= Mixer2,
	Execute					:= n_Step = 20 OR n_Step = 200);

END_FUNCTION_BLOCK

// ---- POUs/FB_SetOutputDataToIO.TcPOU
FUNCTION_BLOCK FB_SetOutputDataToIO
VAR_INPUT
	// Mixer 
	b_MI1_set_run: BOOL;
	b_Ml1_Enable : BOOL;
	b_MI1_Curved_Speed_On : BOOL;
	f_MI1_Override_Speed :REAL;
	f_MI1_Override_Max_Speed :REAL;
	
	
	// Concrete Pump
	b_CP1_Forward_On : BOOL;
	b_CP1_Backward_On : BOOL;
	b_CP1_Flush_On :BOOL;	
	b_CP1_Check_On : BOOL;
	n_CP_Flowrate_mode : BOOL;
	n_CP1_Operate_Flowrate : UDINT;
	n_CP1_Check_Flowrate : UDINT;	
	n_CP1_Flush_Flowrate : UDINT;	
	f_dosing_volume:INT;
	
	n_CP1_max_speed : INT;  // rpm
	n_CP1_target_speed: INT; // rpm

	// Admixture pump (High)
	b_AP1_Power_On : BOOL;
	b_AP1_Run : BOOL;
	b_AP1_Flush_On :BOOL;
	b_AP1_Check_On :BOOL;
	
	n_AP1_Flowrate_mode : BOOL;
	n_AP1_Max_Flowrate : INT;
	n_AP1_Operate_Flowrate : UDINT;
	n_AP1_Check_Flowrate : UDINT;
	n_AP1_Flush_Flowrate : UDINT;
	n_AP1_Dosing_factor : INT;
	
	// Admixture pump (High)
	b_SP1_Power_On : BOOL;
	b_SP1_Run : BOOL;
	b_SP1_Flush_On :BOOL;
	b_SP1_Check_On :BOOL;
	
	n_SP1_Flowrate_mode : BOOL;
	n_SP1_Max_Flowrate : INT;
	n_SP1_Operate_Flowrate : UDINT;
	n_SP1_Check_Flowrate : UDINT;
	n_SP1_Flush_Flowrate : UDINT;
	n_SP1_Dosing_factor : INT;
	
END_VAR
VAR_OUTPUT
END_VAR
VAR	
	// Condition
	_b_Condition_M11 : BOOL;
	_n_Step_M11 : INT;
	
	_n_temp_flowrate_CP1 : UDINT; 
	_n_temp_speed_CP1: INT;
	_n_temp_speed_AP1 : UDINT;
	_n_temp_speed_SP1 : UDINT;
	
	_n_temp_speed_MI1 : INT;
END_VAR

// ***********************************************************************************
//
// Müller-steinag Gruppe, Kandergrien Einigen, CH-3646 Bern
// ETH Zurich, Building HIF E26, Laura-Hezner-Weg 7, CH-8093 Zürich
// 
// ***********************************************************************************
// 
// PROJECT     :  A061 Digital Casting System 
// FUNCTION    :  Set data to IO the process
// AUTHOR      :  Weiting Chen
// EMAIL       :  chenw@usi.ch
// Copyright   :  USI Mendrisio; ETH Zürich; Müller-steinag Gruppe (CH) 2023
// Contributor :  Philippe Fleischmann
//
// ***********************************************************************************


//***********************************************************************************
// MI1 
//***********************************************************************************

IF b_MI1_Curved_Speed_On THEN
		// run curved Speed mode
		P_MI1_Curved_Speed();
		P_MI1_Curved_Speed.b_set_run := b_MI1_set_run;
		P_MI1_Curved_Speed.b_check_mode_on:= b_MI1_Curved_Speed_On;
		_n_temp_speed_MI1:=F_ScalAnalogOut(
			n_Input:= REAL_TO_INT(P_MI1_Curved_Speed.f_MI1_speed),
			n_InMin:= 0, 
			n_InMax:= 120, 
			n_OutMin:= 0, 
			n_OutMax:= 100);
ELSE
	_n_temp_speed_MI1:=F_ScalAnalogOut(
		n_Input:= REAL_TO_INT(f_MI1_Override_Speed),
		n_InMin:= 0, 
		n_InMax:= 120, 
		n_OutMin:= 0, 
		n_OutMax:= 100);
END_IF
GVL.n_MI1_OverrideSpeed:=_n_temp_speed_MI1;

// ***********************************************************************************
// Concrete Pump 1 
// ***********************************************************************************


// Start
IF  P_CP1_Enable.n_Step=20 THEN
	GVL_IO.ob_CP1_Start:=TRUE;
ELSE
	GVL_IO.ob_CP1_Start:=FALSE;
END_IF

// Stop
IF  P_CP1_Enable.n_Step=40 THEN
	GVL_IO.ob_CP1_Stop:=TRUE;
ELSE
	GVL_IO.ob_CP1_Stop:=FALSE;
END_IF

GVL_IO.ob_CP1_Forward := b_CP1_Forward_On; // Forward
GVL_IO.ob_CP1_Backward := b_CP1_Backward_On; // Backward

// Set speed for pump
IF b_CP1_Flush_On THEN
	//
	// Process speed for flushing or filling the pipe
	 _n_temp_flowrate_CP1:=n_CP1_Flush_Flowrate;
ELSIF P_CP1_Check.n_Step=20 OR P_CP1_Check.n_Step=25 THEN
	//	
	// Check Flowrate for pump
	_n_temp_flowrate_CP1 :=n_CP1_Check_Flowrate;
ELSE
	//
	// Process speed for pump
	_n_temp_flowrate_CP1 :=n_CP1_Operate_Flowrate;
END_IF


// Concrete pump speed  0 (0V) to 75 rpm (10V)
IF NOT n_CP_Flowrate_mode THEN
	// set from rpm
	GVL_IO.on_CP1_Speed:=F_ScalAnalogOut(
		n_Input:= INT_TO_UDINT(n_CP1_target_speed),
		n_InMin:= 0, 
		n_InMax:= INT_TO_UDINT(n_CP1_max_speed), 
		n_OutMin:= 0, 
		n_OutMax:= 32767);
ELSE
	// set from flowrate
	GVL_IO.on_CP1_Speed:=F_ScalAnalogOut(
		n_Input:= _n_temp_flowrate_CP1,
		n_InMin:= 0, 
		n_InMax:= INT_TO_UDINT(n_CP1_max_speed*f_dosing_volume), 
		n_OutMin:= 0, 
		n_OutMax:= 32767);
END_IF


//***********************************************************************************
// AP1 (High dosage)
//***********************************************************************************

// Power on
GVL_IO.ob_AP1_Power_On := b_AP1_Power_On;
// Pressure okey always set to true
GVL_IO.ob_AP1_Pressure_Ok := TRUE;
// Bucket not empty always set to true
GVL_IO.ob_AP1_Not_Empty := TRUE;
// Pulse a preset amount not in use
GVL_IO.ob_AP1_Pulse := FALSE;

// Start pump
IF 	   P_AP1_OnOff.n_Step=30 
	OR P_AP1_Check.n_Step=30
THEN
	//
	// Pump on
	GVL_IO.ob_AP1_Start:=TRUE;
ELSE
	//
	// Pump off
	GVL_IO.ob_AP1_Start:=FALSE;
END_IF

//
// Set speed for pump
IF b_AP1_Flush_On AND P_AP1_OnOff.n_Step=30 THEN
	//
	// Process speed for flushing the pipe
	_n_temp_speed_AP1:=n_AP1_Flush_Flowrate;
ELSIF P_AP1_Check.n_Step=20 OR P_AP1_Check.n_Step=30 THEN
	//	
	// Check Flowrate for pump
	_n_temp_speed_AP1:=n_AP1_Check_Flowrate;
ELSE
	//
	// Process speed for pump
	_n_temp_speed_AP1:=n_AP1_Operate_Flowrate;
END_IF

GVL_IO.on_AP1_Speed:=F_ScalAnalogOut(
	n_Input:= _n_temp_speed_AP1,
	n_InMin:= 0, 
	n_InMax:= INT_TO_UDINT(n_AP1_Max_Flowrate)*n_AP1_Dosing_factor, 
	n_OutMin:= 0, 
	n_OutMax:= 32767);

//***********************************************************************************
// SP1 (Low dosage)
//***********************************************************************************

// Power on
GVL_IO.ob_SP1_Power_On := b_SP1_Power_On;
// Pressure okey always set to true
GVL_IO.ob_SP1_Pressure_Ok := TRUE;
// Bucket not empty always set to true
GVL_IO.ob_SP1_Not_Empty := TRUE;
// Pulse a preset amount not in use
GVL_IO.ob_SP1_Pulse := FALSE;

// Start pump
IF		P_SP1_OnOff.n_step= 30 
	OR 	P_SP1_Check.n_Step= 30 
THEN
	//
	// Pump On
	GVL_IO.ob_SP1_Start:=TRUE;
ELSE
	//
	// Pump On
	GVL_IO.ob_SP1_Start:=FALSE;
END_IF

//
// Set speed for pump
IF b_SP1_Flush_On AND P_SP1_OnOff.n_Step=30 THEN
	//
	// Process speed for flushing the pipe
	_n_temp_speed_SP1:=n_SP1_Flush_Flowrate;
ELSIF P_SP1_Check.n_Step=20 OR P_SP1_Check.n_Step=30 THEN
	//	
	// Check Flowrate for pump
	_n_temp_speed_SP1:=n_SP1_Check_Flowrate;
ELSE
	//
	// Process speed for pump
	_n_temp_speed_SP1:=n_SP1_Operate_Flowrate;
END_IF

GVL_IO.on_SP1_Speed:=F_ScalAnalogOut(
	n_Input:= _n_temp_speed_SP1,
	n_InMin:= 0, 
	n_InMax:= INT_TO_UDINT(n_SP1_Max_Flowrate)*n_SP1_Dosing_factor, 
	n_OutMin:= 0, 
	n_OutMax:= 32767);

END_FUNCTION_BLOCK

// ---- POUs/Utils/F_ScalAnalogOut.TcPOU
FUNCTION F_ScalAnalogOut : INT
VAR_INPUT
	n_Input:UDINT;
	n_InMin:UDINT;
	n_InMax:UDINT;
	n_OutMin:UDINT;
	n_OutMax:UDINT;

END_VAR
VAR
	f_Input:REAL;
	f_InMin:REAL;
	f_InMax:REAL;
	f_OutMin:REAL;
	f_OutMax:REAL;
	f_DeltaIn:REAL;
	f_DeltaOut:REAL;
END_VAR

//
// Convert integer to real 
f_Input:=UDINT_TO_REAL(n_Input);
f_InMin:=UDINT_TO_REAL(n_InMin);
f_InMax:=UDINT_TO_REAL(n_InMax);
f_OutMin:=UDINT_TO_REAL(n_OutMin);
f_OutMax:=UDINT_TO_REAL(n_OutMax);

//
// Check plausibility 

IF f_Input > f_InMax THEN
	f_Input := f_InMax;
END_IF

IF f_InMax = f_InMin THEN	
	//
	// Not plausible output fix value
	F_ScalAnalogOut := 0;
ELSE
	// Check the input data is lager than maximum
	IF f_Input > f_InMax THEN
		f_Input := f_InMax;
	END_IF
	//
	// Plausible calculate output 
	f_DeltaIn:=f_InMax-f_InMin;
	f_DeltaOut:=f_OutMax-f_OutMin;
	F_ScalAnalogOut :=REAL_TO_INT((f_DeltaOut/f_DeltaIn)*(f_Input-f_InMin));	
END_IF

END_FUNCTION

// ---- POUs/Component/P_CP1_Check.TcPOU
PROGRAM P_CP1_Check
VAR_INPUT
	n_Step: INT := 0;	
	b_set_run : BOOL;
	b_check_mode_on : BOOL;
	t_check_duration :TIME;
END_VAR
VAR
	//
	// BOOL 
	b_Condition: BOOL;
	b_No_Emergency_Stop:BOOL :=TRUE;
	
	//
	// Timer 
	t_CP1_Check_Time: TON;
	//
	t_CP1_Puls_Enable: TON;	
	t_CP1_Puls_Disable: TON;	
	
END_VAR

// ***********************************************************************************
//
// Müller-steinag Gruppe, Kandergrien Einigen, CH-3646 Bern
// ETH Zurich, Building HIF E26, Laura-Hezner-Weg 7, CH-8093 Zürich
// 
// ***********************************************************************************
// 
// PROJECT     :  A061 Digital Casting System 
// FUNCTION    :  Step chain for Concrete pump calibration
// AUTHOR      :  Weiting Chen
// EMAIL       :  chenw@usi.ch
// Copyright   :  USI Mendrisio; ETH Zürich; Müller-steinag Gruppe (CH) 2023
// Contributor :  Philippe Fleischmann
//
// ***********************************************************************************

// Ignore emergency stop
b_No_Emergency_Stop:=TRUE;

//
// Initalization
IF n_Step=0 THEN
	//
	// Check condition 
	b_Condition:=TRUE;
	//
	// Do step
	IF b_Condition THEN
		b_Condition:=FALSE;
		n_Step:=10;
	END_IF
END_IF

//
// Check grid mounted and no errors and the check mode on 
IF n_Step=10 THEN
	//
	// Check condition 
	b_Condition:= GVL_IO.ib_CP1_Ready AND GVL_IO.ib_CP1_Safety_Grid_Mounted AND NOT GVL_IO.ib_CP1_Drive_Error;
	//
	// Do step
	IF b_Condition AND b_No_Emergency_Stop THEN
		b_Condition:=FALSE;
		n_Step:=20;
	END_IF
END_IF

//
// Send enable to pump and wait for start 
IF n_Step=20 THEN
	//
	// Check condition 
	b_Condition:= b_check_mode_on AND b_set_run;
	//
	// Do step
	IF b_Condition AND b_No_Emergency_Stop THEN
		b_Condition:=FALSE;
		n_Step:=25;
	END_IF
END_IF

//
// Pump enabled checking for errors or grid removed
IF n_Step=25 THEN
	//
	// Check condition 
	b_Condition:= t_CP1_Check_Time.Q;
	//
	// Do step
	IF b_Condition THEN
		b_Condition:=FALSE;
		n_Step:=30;
	END_IF
END_IF

//
// Pump enabled checking for errors or grid removed
IF n_Step=30 THEN
	//
	// Check condition 
	b_Condition:= TRUE;
	//
	// Do step
	IF b_Condition THEN
		b_Condition:=FALSE;
		n_Step:=40;
	END_IF
END_IF

//
// 
IF n_Step=40 THEN
	//
	// Check condition 
	b_Condition:=TRUE;
	//
	// Do step
	IF b_Condition AND b_No_Emergency_Stop THEN
		b_Condition:=FALSE;
		n_Step:=50;
	END_IF
END_IF

//
// Return to step 10 
IF n_Step=50 THEN
	//
	// Check condition 
	b_Condition:=TRUE;
	//
	// Do step
	IF b_Condition THEN
		//
		//Reset 
		b_set_run:=FALSE;
		b_check_mode_on:=FALSE;
		b_Condition:=FALSE;
		n_Step:=10;
	END_IF
END_IF

// ****************************************
// Timer
// ****************************************
t_CP1_Check_Time(
	IN:=n_Step=25,
	PT:=t_check_duration);

// ****************************************
// Reset
// ****************************************
IF NOT b_check_mode_on THEN
  //
  // Rest step chain
  n_Step:=0;
END_IF

END_PROGRAM

// ---- POUs/FB_GetOutputData.TcPOU
FUNCTION_BLOCK FB_GetOutputData
VAR_INPUT
	//Gerenal
	b_Output_number_REALMode : BOOL;
END_VAR
VAR_IN_OUT
	//CC1
	b_mode_manual : BOOL;
	b_mode_laptop : BOOL; 	
	b_mode_robot : BOOL; 
	b_CC1_power_on : BOOL; 
	n_current_mode : INT;

	//MI1
	b_MI1_Is_Run:BOOL;
	b_MI1_is_ready : BOOL;
	n_MI1_status_SpeedM1 : INT;
	n_MI1_status_SpeedM2 : INT;
	f_Status_Torque_Motor_1 : REAL;
	f_Status_Torque_Motor_2 : REAL;
	f_MI1_status_temperature_funnel_outlet : REAL; 		
	f_MI1_status_Pressure_funnel_inlet : REAL; 	
	f_MI1_status_temperature_motor_1 : REAL; 			 
	f_MI1_status_temperature_motor_2 : REAL; 			

	//CP1
	b_CP1_is_run : BOOL;
	b_CP1_is_ready : BOOL;
	b_CP1_power_on :BOOL;
	b_CP1_safety_grid_on : BOOL;
	b_CP1_drive_error :BOOL;
	
	f_CP1_status_temperature_concrete_fresh : REAL; // [°C]
	f_CP1_status_temperature_Concrete_pump : REAL; // [°C] 
	f_CP1_status_pressure_Concrete_pump: REAL; // [bar]
	
	//AP1
	b_AP1_is_run : BOOL;
	b_AP1_is_ready : BOOL;
	b_AP1_no_error : BOOL;
	
	//SP1
	b_SP1_is_run : BOOL;
	b_SP1_is_ready : BOOL;
	b_SP1_no_error : BOOL;
	
END_VAR
VAR_OUTPUT

END_VAR
VAR
	tempVelo_M1 : LREAL;
	tempVelo_M2 : LREAL;
END_VAR

// ***********************************************************************************
//
// Müller-steinag Gruppe, Kandergrien Einigen, CH-3646 Bern
// ETH Zurich, Building Hin E26, Laura-Hezner-Weg 7, CH-8093 Zürich
// 
// ***********************************************************************************
// 
// PROJECT     :  A061 Digital Casting System 
// FUNCTION    :  Read data from IO and process 
// AUTHOR      :  Weiting Chen
// EMAIL       :  chenw@usi.ch
// Copyright   :  USI Mendrisio; ETH Zürich; Müller-steinag Gruppe (CH) 2024
// Contributor :  Seyma Gürel / Philippe Fleischmann 
//
// ***********************************************************************************

b_mode_manual := GVL.b_mode_manual;
b_mode_laptop := GVL.b_mode_laptop; 	
b_mode_robot := GVL.b_mode_robot; 
b_CC1_power_on := GVL.b_CC1_power_on; 

IF GVL.s_current_mode = 'Controller'THEN
	n_current_mode := 1;
ELSIF GVL.s_current_mode = 'Laptop' THEN
	n_current_mode := 2;
ELSIF GVL.s_current_mode = 'Robot' THEN
	n_current_mode := 3;
ELSE 
	n_current_mode := 4;
END_IF

//// Mixer 1_2 
//Status
b_MI1_Is_Run := GVL.b_MI1_Is_Run;
b_MI1_is_ready := GVL.b_MI1_ReadToDrive;

//current speed [rpm]
tempVelo_M1 := ABS(GVL.Axis_Mixer1.NcToPlc.ActVelo/6);  // velocity to rpm
GVL.f_MI1_ActSpeedM1 := LREAL_TO_INT(tempVelo_M1);
n_MI1_status_SpeedM1 := GVL.f_MI1_ActSpeedM1 ;

tempVelo_M2 := ABS(GVL.Axis_Mixer2.NcToPlc.ActVelo/6);  // velocity to rpm
GVL.f_MI1_ActSpeedM2 := LREAL_TO_INT(tempVelo_M2);
n_MI1_status_SpeedM2 := GVL.f_MI1_ActSpeedM2 ;

//Torque
GVL.f_MID1_ActCurrent:=GVL_IO.in_MID1_ActAbsCurrent * 5.9 / 1000;
GVL.f_MID1_ActTorque:=GVL.f_MID1_ActCurrent * 0.8 * 8; // Torque constante / Gear transaltion 
f_Status_Torque_Motor_1:= GVL.f_MID1_ActTorque;

GVL.f_MID2_ActCurrent:=GVL_IO.in_MID2_ActAbsCurrent * 5.9 / 1000;
GVL.f_MID2_ActTorque:=GVL.f_MID2_ActCurrent * 0.8 * 8; // Torque constante / Gear transaltion
f_Status_Torque_Motor_2:= GVL.f_MID2_ActTorque;

//Temperature
IF b_Output_number_REALMode THEN
	f_MI1_status_temperature_funnel_outlet := F_LowpassFilter(GVL_IO.in_Temp_Funnel_Outlet) * 0.1; 
	f_MI1_status_temperature_motor_1 := F_LowpassFilter(UINT_TO_REAL(GVL_IO.in_MID1_ActMotorTemperature)) * 0.1;
	f_MI1_status_temperature_motor_2 := F_LowpassFilter(UINT_TO_REAL(GVL_IO.in_MID2_ActMotorTemperature)) * 0.1;
ELSE
	f_MI1_status_temperature_funnel_outlet := F_LowpassFilter(GVL_IO.in_Temp_Funnel_Outlet); 
	f_MI1_status_temperature_motor_1 := F_LowpassFilter(UINT_TO_REAL(GVL_IO.in_MID1_ActMotorTemperature));
	f_MI1_status_temperature_motor_2 := F_LowpassFilter(UINT_TO_REAL(GVL_IO.in_MID2_ActMotorTemperature));
END_IF

//Pressure TODO
//f_CP1_status_pressure_Concrete_pump := F_DecimalData(GVL_RESD.f_CP1_status_pressure_Concrete_pump, 3, TRUE),	
f_MI1_status_Pressure_funnel_inlet := (INT_TO_REAL(GVL_IO.in_Pressure_Funnel)/32767)*40;


////Concrete Pump 	
//Status
GVL.b_CP1_Is_Run := GVL_IO.ob_CP1_Forward;
b_CP1_is_run := GVL.b_CP1_Is_Run;

GVL.b_CP1_is_ready := GVL_IO.ib_CP1_Ready;
b_CP1_is_ready := GVL.b_CP1_is_ready;


GVL.b_CP1_power_on :=  GVL_IO.ib_CP1_Ready;
b_CP1_power_on := GVL.b_CP1_power_on;

GVL.b_CP1_safety_grid_on := GVL_IO.ib_CP1_Safety_Grid_Mounted;
b_CP1_safety_grid_on := GVL.b_CP1_safety_grid_on;
	
GVL.b_CP1_drive_error := GVL_IO.ib_CP1_Drive_Error;
b_CP1_drive_error := GVL.b_CP1_drive_error;


//Torque
//Temperature
IF b_Output_number_REALMode THEN
	f_CP1_status_temperature_concrete_fresh := F_LowpassFilter(GVL_IO.in_Temp_CPump_fresh)*0.1;
	f_CP1_status_temperature_Concrete_pump := F_LowpassFilter(GVL_IO.in_Temp_CPump)*0.1; 
ELSE
	f_CP1_status_temperature_concrete_fresh := F_LowpassFilter(GVL_IO.in_Temp_CPump_fresh);
	f_CP1_status_temperature_Concrete_pump := F_LowpassFilter(GVL_IO.in_Temp_CPump); 
END_IF

//Pressure

f_CP1_status_pressure_Concrete_pump:= (INT_TO_REAL(GVL_IO.in_Pressure_Pump)/32767)*40;



////AP1
//Status
b_AP1_is_run := GVL.b_AP1_Is_Run;

GVL.b_AP1_is_ready := GVL_IO.ib_AP1_Ready;
b_AP1_is_ready := GVL.b_AP1_is_ready;

GVL.b_AP1_no_error := GVL_IO.ib_AP1_No_Error;
b_AP1_no_error := GVL.b_AP1_no_error;

//f_AP1_max_flowrate := GVL.n_AP1_Max_Flowrate;						

////SP1
//Status
b_SP1_is_run := GVL.b_SP1_Is_Run;

GVL.b_SP1_is_ready := GVL_IO.ib_SP1_Ready;
b_SP1_is_ready := GVL.b_SP1_is_ready;

GVL.b_SP1_no_error := GVL_IO.ib_SP1_No_Error;
b_SP1_no_error := GVL.b_SP1_no_error;

//f_SP1_max_flowrate := GVL.n_SP1_Max_Flowrate;

END_FUNCTION_BLOCK

// ---- POUs/P_PNDataConvert.TcPOU
PROGRAM P_PNDataConvert
VAR
	
	sizearr: UINT;

	arr_GISlot: ARRAY[32..255] OF BYTE;
	arr_GOSlot: ARRAY[32..255] OF BYTE;

	arr_CC1_DOSlot: ARRAY[0..7] OF BOOL;
	arr_CC1_DISlot: ARRAY[0..7] OF BOOL;
	
	
	arr_MI1_DOSlot: ARRAY [0..7] OF BOOL;
	arr_MI1_DISlot: ARRAY [0..7] OF BOOL;

	arr_CP1_DOSlot: ARRAY [0..7] OF BOOL;
	arr_CP1_DISlot: ARRAY [0..7] OF BOOL;

	arr_AP1_DOSlot: ARRAY [0..7] OF BOOL;
	arr_AP1_DISlot: ARRAY [0..7] OF BOOL;

	arr_SP1_DOSlot: ARRAY [0..7] OF BOOL;
	arr_SP1_DISlot: ARRAY [0..7] OF BOOL;

	// inline mixer
	on_MI1_status_speed_motor_1: UINT;
	on_MI1_status_speed_motor_2: UINT;
	
	on_MI1_status_torque_motor_1: UINT;
	on_MI1_status_torque_motor_2: UINT;
	
	on_MI1_status_temperature_motor_1 : UINT; 			
	on_MI1_status_temperature_motor_2 : UINT;
	
	on_MI1_status_temperature_funnel_outlet : UINT; 
	on_MI1_status_Pressure_funnel_inlet: UINT;
	on_CP1_status_temperature_concrete_fresh : UINT;
	on_CP1_status_temperature_Concrete_pump : UINT;
	on_CP1_status_pressure_Concrete_pump : UINT;
END_VAR

// ***********************************************************************************
//
// Müller-steinag Gruppe, Kandergrien Einigen, CH-3646 Bern
// ETH Zurich, Building HIF E26, Laura-Hezner-Weg 7, CH-8093 Zürich
//
// ***********************************************************************************
//
// PROJECT: A061 Digital Casting System
// FUNCTION: Profinet Variable Convertor
// AUTHOR: Weiting Chen
// EMAIL: chenw@usi.ch
// Copyright: USI Mendrisio; ETH Zürich; Müller-steinag Gruppe (CH) 2024
//
// ***********************************************************************************

// output(o_) to robot digital input (DI); input(i_) from robot digital output(DO)

// Array of DO_From_ROB is 0 to 255 bits | 0 to 31 bytes
// Array of GO_From_ROB is 256 to 2047 bits | 32 to 255 bytes
// Array of DI_To_ROB is 0 to 255 bits | 0 to 31 bytes
// Array of GI_To_ROB is 256 to 2047 bits | 32 to 255 bytes

// scale data by 100 for Real to UINT 
// Group input and output slots
	MEMCPY(ADR(GVL_PN.GI_To_ROB), ADR(arr_GISlot), SIZEOF(arr_GOSlot));
	MEMCPY(ADR(arr_GOSlot), ADR(GVL_PN.GO_From_ROB), SIZEOF(arr_GOSlot));
	
// Concrete Controller *****
	// Digital output from robot( mapping from 0 to 7 in robotstudio)
		arr_CC1_DOSlot := F_CONVERT_BYTE_TO_BIT(GVL_PN.DO_From_ROB[0]);
		GVL_ROB.ib_CC1_enable := arr_CC1_DOSlot[0]; // #0
		GVL_ROB.ib_CC1_reset := arr_CC1_DOSlot[1]; // #1
		GVL_ROB.ib_CC1_data_recording := arr_CC1_DOSlot[2]; // #2
		
	// Group output from Robot ( mapping from 32 to 46, 8*2Bytes in robotstudio)
		F_Convert_2Byte_to_Int(GVL_ROB.in_spare, arr_GOSlot[32], arr_GOSlot[33]); // #256 to 271

	// Digital input to robot (mapping from 0 to 7 in robotstudio)
		arr_CC1_DISlot[0] := GVL_ROB.ob_mode_manual; // #0
		arr_CC1_DISlot[1] := GVL_ROB.ob_mode_laptop;
		arr_CC1_DISlot[2] := GVL_ROB.ob_mode_robot;
		arr_CC1_DISlot[3] := GVL_ROB.ob_CC1_power_on;
		
		// pointer 
		MEMCPY(ADR(GVL_PN.DI_To_ROB[0]), ADR(arr_CC1_DISlot), SIZEOF(arr_CC1_DISlot));
	
		
	// Group Input To Robot (32 to 46; 8*2Bytes)
		F_Convert_Int_to_2Byte(GVL_ROB.on_current_mode, arr_GISlot[32], arr_GISlot[33]); // #256 to 271


// Inline Mixer (MI1) *****
	// Digital output from robot ( mapping from 8 to 15 in robotstudio)
		arr_MI1_DOSlot := F_CONVERT_BYTE_TO_BIT(GVL_PN.DO_From_ROB[1]);
		GVL_ROB.ib_MI1_set_run := arr_MI1_DOSlot[0]; // [0 rpm to 120 rpm]
		GVL_ROB.ib_MI1_enable := arr_MI1_DOSlot[1];
		GVL_ROB.ib_MI1_set_curved_speed_mode_on := arr_MI1_DOSlot[2];

	// Group output from Robot ( mapping from 47 to 61, 8*2Bytes in robotstudio)
		//F_Convert_2Byte_to_Int(GVL_ROB.in_MI1_set_speed, arr_GOSlot[47], arr_GOSlot[48]);
		// 
		F_Convert_2Byte_to_Uint(GVL_ROB.in_MI1_set_speed, arr_GOSlot[47], arr_GOSlot[48]); // 376-391
		
		
	// Digital input to robot (mapping from 8 to 15 in robotstudio)
		//arr_MI1_DISlot := F_CONVERT_BYTE_TO_BIT(GVL_PN.DI_To_ROB[1]);
		arr_MI1_DISlot[0] := GVL_ROB.ob_MI1_is_run;
		arr_MI1_DISlot[1] := GVL_ROB.ob_MI1_is_ready;
		
		// pointer 
		MEMCPY(ADR(GVL_PN.DI_To_ROB[1]), ADR(arr_MI1_DISlot), SIZEOF(arr_MI1_DISlot));

	// Group Input To Robot (mapping from 47 to 76, 16*2Bytes in robotstudio)
		
		// data convert 
		on_MI1_status_speed_motor_1:=REAL_TO_UINT(INT_TO_REAL(GVL_ROB.on_MI1_status_speed_motor_1));
		on_MI1_status_speed_motor_2:=REAL_TO_UINT(INT_TO_REAL(GVL_ROB.on_MI1_status_speed_motor_2));
		
		on_MI1_status_torque_motor_1:=REAL_TO_UINT(GVL_ROB.on_MI1_status_torque_motor_1*100);
		on_MI1_status_torque_motor_2:=REAL_TO_UINT(GVL_ROB.on_MI1_status_torque_motor_2*100);
		
		on_MI1_status_temperature_motor_1:=REAL_TO_UINT(GVL_ROB.on_MI1_status_temperature_motor_1);
		on_MI1_status_temperature_motor_2:=REAL_TO_UINT(GVL_ROB.on_MI1_status_temperature_motor_2);
		
		on_MI1_status_temperature_funnel_outlet:=REAL_TO_UINT(GVL_ROB.on_MI1_status_temperature_funnel_outlet);
		on_MI1_status_pressure_funnel_inlet:=REAL_TO_UINT(GVL_ROB.on_MI1_status_pressure_funnel_inlet*100);		
		
		
		F_Convert_Uint_to_2Byte(on_MI1_status_speed_motor_1, arr_GISlot[47], arr_GISlot[48]);
		F_Convert_Uint_to_2Byte(on_MI1_status_speed_motor_2, arr_GISlot[49], arr_GISlot[50]);
		
		F_Convert_Uint_to_2Byte(on_MI1_status_torque_motor_1, arr_GISlot[51], arr_GISlot[52]);
		F_Convert_Uint_to_2Byte(on_MI1_status_torque_motor_2, arr_GISlot[53], arr_GISlot[54]);
		F_Convert_Uint_to_2Byte(on_MI1_status_temperature_motor_1, arr_GISlot[55], arr_GISlot[56]);
		F_Convert_Uint_to_2Byte(on_MI1_status_temperature_motor_2, arr_GISlot[57], arr_GISlot[58]);
		F_Convert_Uint_to_2Byte(on_MI1_status_temperature_funnel_outlet, arr_GISlot[59], arr_GISlot[60]);
		F_Convert_Uint_to_2Byte(on_MI1_status_Pressure_funnel_inlet, arr_GISlot[61], arr_GISlot[62]);	

// Concrete pump (CP1) *****
	// Digital output from robot (mapping from 16 to 23 in robotstudio )
		arr_CP1_DOSlot := F_CONVERT_BYTE_TO_BIT(GVL_PN.DO_From_ROB[2]);
		GVL_ROB.ib_CP1_forward_on := arr_CP1_DOSlot[0]; // #16
		GVL_ROB.ib_CP1_backward_on := arr_CP1_DOSlot[1];		// 241219 Backward is not working from the conctroller
		GVL_ROB.ib_CP1_check_on := arr_CP1_DOSlot[2];
		GVL_ROB.ib_CP1_flush_on := arr_CP1_DOSlot[3];

	// Group output from Robot ( mapping from 62 to 76, 8*2Bytes in robotstudio)
		F_Convert_2Byte_to_Uint(GVL_ROB.in_CP1_set_speed, arr_GOSlot[62], arr_GOSlot[63]); // 0 to 75 [rpm] #496
		F_Convert_2Byte_to_Uint(GVL_ROB.in_CP1_set_flowrate, arr_GOSlot[64], arr_GOSlot[65]); // 0 to 16 [l/min]
		F_Convert_2Byte_to_Uint(GVL_ROB.in_CP1_set_dosing_volume, arr_GOSlot[66], arr_GOSlot[67]); 	// calibration in 230926 WT 0.32
		F_Convert_2Byte_to_Uint(GVL_ROB.in_CP1_set_check_Flowrate, arr_GOSlot[68], arr_GOSlot[69]);	// [l/min]
		F_Convert_2Byte_to_Uint(GVL_ROB.in_CP1_concrete_density, arr_GOSlot[70], arr_GOSlot[71]); // [g/ml]
		F_Convert_2Byte_to_Uint(GVL_ROB.in_CP1_concrete_mass, arr_GOSlot[72], arr_GOSlot[73]); // [g]
		F_Convert_2Byte_to_Uint(GVL_ROB.in_CP1_set_flush_flowrate, arr_GOSlot[74], arr_GOSlot[75]); // [l/min]
		// F_Convert_2Byte_to_Uint(GVL_ROB.t_CP1_set_check_duration, arr_GOSlot[76], arr_GOSlot[77]);	 check with 32 bit


	// Digital input to robot (mapping from 16 to 23 in robotstudio)
		//arr_CP1_DISlot := F_CONVERT_BYTE_TO_BIT(GVL_PN.DI_To_ROB[2]);
		arr_CP1_DISlot[0] := GVL_ROB.ob_CP1_is_run;		// #16
		arr_CP1_DISlot[1] := GVL_ROB.ob_CP1_is_ready;	// #17
		arr_CP1_DISlot[2] := GVL_ROB.ob_CP1_power_on;	// #18
		arr_CP1_DISlot[3] := GVL_ROB.ob_CP1_safety_grid_on;
		arr_CP1_DISlot[4] := GVL_ROB.ob_CP1_drive_error;
		
		
		MEMCPY(ADR(GVL_PN.DI_To_ROB[2]), ADR(arr_CP1_DISlot), SIZEOF(arr_CP1_DISlot));

	// Group Input To Robot (mapping from 77 to 91, 8*2Bytes in robotstudio)
		on_CP1_status_temperature_concrete_fresh := REAL_TO_UINT(GVL_ROB.on_CP1_status_temperature_concrete_fresh);
		on_CP1_status_temperature_Concrete_pump := REAL_TO_UINT(GVL_ROB.on_CP1_status_temperature_concrete_pump);
		on_CP1_status_pressure_Concrete_pump := REAL_TO_UINT(GVL_ROB.on_CP1_status_pressure_concrete_pump*100);

		F_Convert_Uint_to_2Byte(on_CP1_status_temperature_concrete_fresh, arr_GISlot[77], arr_GISlot[78]); // [°C] #624-639
		F_Convert_Uint_to_2Byte(on_CP1_status_temperature_Concrete_pump, arr_GISlot[79], arr_GISlot[80]); // [°C]
		F_Convert_Uint_to_2Byte(on_CP1_status_pressure_Concrete_pump, arr_GISlot[81], arr_GISlot[82]); // [ bar]

// Admixture pump, High dosage ViscoTech Pump *****
	// Digital output from robot (mapping from 24 to 31 in robotstudio )
		arr_AP1_DOSlot := F_CONVERT_BYTE_TO_BIT(GVL_PN.DO_From_ROB[3]);
		GVL_ROB.ib_AP1_set_run := arr_AP1_DOSlot[0]; // #24
		GVL_ROB.ib_AP1_check_on := arr_AP1_DOSlot[1];
		GVL_ROB.ib_AP1_flush_on := arr_AP1_DOSlot[2];
		GVL_ROB.ib_AP1_power_on := arr_AP1_DOSlot[3];
		

	// Group output from Robot ( mapping from 77 to 91, 8*2Bytes in robotstudio)
		F_Convert_2Byte_to_Uint(GVL_ROB.in_AP1_set_flowrate, arr_GOSlot[78], arr_GOSlot[79]); // **** [ml/min] #77
		F_Convert_2Byte_to_Uint(GVL_ROB.in_AP1_set_dosing_factor, arr_GOSlot[80], arr_GOSlot[81]);
		
		F_Convert_2Byte_to_Uint(GVL_ROB.in_AP1_set_check_flowrate, arr_GOSlot[82], arr_GOSlot[83]);
		F_Convert_2Byte_to_Uint(GVL_ROB.in_AP1_material_density, arr_GOSlot[84], arr_GOSlot[85]);
		F_Convert_2Byte_to_Uint(GVL_ROB.in_AP1_material_mass, arr_GOSlot[86], arr_GOSlot[87]);
		F_Convert_2Byte_to_Uint(GVL_ROB.in_AP1_set_flush_flowrate, arr_GOSlot[88], arr_GOSlot[89]);
		// F_Convert_2Byte_to_Int(GVL_ROB.t_AP1_set_check_duration, arr_GOSlot[90], arr_GOSlot[92]); check with 32 bit

	// Digital input to robot (mapping from 24 to 31 in robotstudio)
		//arr_AP1_DISlot := F_CONVERT_BYTE_TO_BIT(GVL_PN.DI_To_ROB[3]);
		arr_AP1_DISlot[0] := GVL_ROB.ob_AP1_is_run; //#24
		arr_AP1_DISlot[1] := GVL_ROB.ob_AP1_is_ready;
		arr_AP1_DISlot[2] := GVL_ROB.ob_AP1_no_error;
		
		
		MEMCPY(ADR(GVL_PN.DI_To_ROB[3]), ADR(arr_AP1_DISlot), SIZEOF(arr_AP1_DISlot));
		
	// Group Input To Robot (mapping from 92 to 106, 8*2Bytes in robotstudio)
		F_Convert_Uint_to_2Byte(GVL_ROB.on_AP1_max_flowrate, arr_GOSlot[92], arr_GOSlot[93]); // [l/min]

// Admixture pump, Low dosage ViscoTech Pump *****
	// Digital output from robot (mapping from 32 to 39 in robotstudio )
		arr_SP1_DOSlot := F_CONVERT_BYTE_TO_BIT(GVL_PN.DO_From_ROB[4]);
		GVL_ROB.ib_SP1_set_run := arr_SP1_DOSlot[0]; // #32
		GVL_ROB.ib_SP1_set_check_on := arr_SP1_DOSlot[1];
		GVL_ROB.ib_SP1_flush_on := arr_SP1_DOSlot[2];
		GVL_ROB.ib_SP1_power_on := arr_SP1_DOSlot[3];

	// Group output from Robot ( mapping from 92 to 106, 8*2Bytes in robotstudio)
		F_Convert_2Byte_to_Uint(GVL_ROB.in_SP1_set_flowrate, arr_GOSlot[94], arr_GOSlot[95]); // **** [ml/min] #92
		F_Convert_2Byte_to_Uint(GVL_ROB.in_SP1_dosing_factor, arr_GOSlot[96], arr_GOSlot[97]);
		
		F_Convert_2Byte_to_Uint(GVL_ROB.in_SP1_set_check_flowrate, arr_GOSlot[98], arr_GOSlot[99]);
		F_Convert_2Byte_to_Uint(GVL_ROB.in_SP1_material_density, arr_GOSlot[100], arr_GOSlot[101]);
		F_Convert_2Byte_to_Uint(GVL_ROB.in_SP1_material_mass, arr_GOSlot[102], arr_GOSlot[103]);
		F_Convert_2Byte_to_Uint(GVL_ROB.in_SP1_flush_flowrate, arr_GOSlot[104], arr_GOSlot[105]);
		
		// F_Convert_2Byte_to_Int(GVL_ROB.t_SP1_Check_Duration, arr_GOSlot[106], arr_GOSlot[107]); // Check with 32 bit

	// Digital input to robot (mapping from 32 to 39 in robotstudio)
		//arr_SP1_DISlot := F_CONVERT_BYTE_TO_BIT(GVL_PN.DI_To_ROB[4]);
		arr_SP1_DISlot[0] := GVL_ROB.ob_SP1_is_run; // #32
		arr_SP1_DISlot[1] := GVL_ROB.ob_SP1_is_ready;
		arr_SP1_DISlot[2] := GVL_ROB.ob_SP1_no_error;
		
		MEMCPY(ADR(GVL_PN.DI_To_ROB[4]), ADR(arr_SP1_DISlot), SIZEOF(arr_SP1_DISlot));

	// Group Input To Robot (mapping from 106 to 120, 8*2Bytes in robotstudio)
		F_Convert_Uint_to_2Byte(GVL_ROB.on_SP1_max_flowrate, arr_GOSlot[106], arr_GOSlot[107]); // [l/min]

(*
// Spare Component *****
	// Digital output from robot (mapping from 40 to .. in robotstudio )
	// Group output from Robot ( mapping from 107 to .., 8*2Bytes in robotstudio)
	// Digital input to robot (mapping from 40 to .. in robotstudio)
	// Group Input To Robot (mapping from 121 to .., 8*2Bytes in robotstudio)
//
*)

END_PROGRAM

// ---- POUs/Utils/F_Convert_2Byte_to_Uint.TcPOU
FUNCTION F_Convert_2Byte_to_Uint 

VAR_IN_OUT
	inputNum : UINT; 
	dataByte1 : BYTE;
	dataByte2 : BYTE;
END_VAR

VAR
	arrByte : ARRAY [0..1] OF BYTE;
END_VAR

arrByte[0]:= dataByte1;
arrByte[1]:= dataByte2;
MEMCPY(ADR(inputNum), ADR(arrByte), 2);

//F_Convert_Int_to_2Byte:=arrByte;

END_FUNCTION

// ---- POUs/Utils/F_Convert_Uint_to_2Byte.TcPOU
FUNCTION F_Convert_Uint_to_2Byte
VAR_IN_OUT
	inputNum : UINT; 
	dataByte1 : BYTE;
	dataByte2 : BYTE;
END_VAR

VAR
	arrByte : ARRAY [0..1] OF BYTE;
END_VAR

MEMCPY(ADR(arrByte), ADR(inputNum), 2);
dataByte1 := arrByte[0];
dataByte2 := arrByte[1];

//F_Convert_Int_to_2Byte:=arrByte;

END_FUNCTION

// ---- POUs/P_Robot_Operate.TcPOU
PROGRAM P_Robot_Operate
VAR
	fb_MC_SetPosition		:FB_SoEAX5000SetPositionOffset;
	pos:LREAL;
	Mixer1_2		: FB_Mixer1_2;
	Analog			: FB_Analog;
	SafetyReset 	: bool;
	b_Enable		: BOOL;
	b_Reset			: BOOL;

	Test : MC_ReadStatus;

	fb_SetOutputDataToIO : FB_SetOutputDataToIO;
	fb_getOutputData : FB_GetOutputData;
	fb_setConfig : FB_SetConfigData;
	
	//
	b_Safety_Reset : BOOL :=FALSE;
	b_Timer_Rest : BOOL;
	t_CC1_Time_Safety_Rest : TIME :=T#5S; //wait 5s for controller restart
	fb_CC1_Trigger_Safety_On : R_TRIG;
	fb_CC1_Trigger_Safety_Off : R_TRIG;
	fb_CC1_Timer_Safety: TON;
	
	

END_VAR

// ***********************************************************************************
//
// Müller-steinag Gruppe, Kandergrien Einigen, CH-3646 Bern
// ETH Zurich, Building HIF E26, Laura-Hezner-Weg 7, CH-8093 Zürich
// 
// ***********************************************************************************
// 
// PROJECT     :  A061 Digital Casting System 
// FUNCTION    :  Robot operate process
// AUTHOR      :  Weiting Chen
// EMAIL       :  chenw@usi.ch
// Copyright   :  USI Mendrisio; ETH Zürich; Müller-steinag Gruppe (CH) 2024
//
// ***********************************************************************************


b_Timer_Rest:=GVL_ROB.ib_CC1_reset;

//controller reset trigger
fb_CC1_Timer_Safety(
					IN:=b_Timer_Rest,
					PT:=t_CC1_Time_Safety_Rest);

fb_CC1_Trigger_Safety_On(clk:=fb_CC1_Timer_Safety.IN);
fb_CC1_Trigger_Safety_Off(clk:=fb_CC1_Timer_Safety.Q);
//b_Safety_Reset:=FALSE;
IF fb_CC1_Trigger_Safety_On.Q THEN
	b_Safety_Reset:=TRUE;
ELSIF
	fb_CC1_Trigger_Safety_Off.Q THEN 
	GVL_ROB.ib_CC1_reset:=FALSE;
	b_Safety_Reset:=FALSE;
END_IF
GVL_IO.ob_CC1_Safety_Reset:= GVL_ROB.ib_CC1_reset OR GVL_IO.ib_CC1_Button_Reset;


// Concrete Conctroller enable 
P_CC1_Enable( b_set_run:= GVL_ROB.ib_CC1_enable);


//***********************************************************************************
// Set Process Configuration
//***********************************************************************************

fb_setConfig(
// Gerenal
// Concrete Controller
// Inline Mixer
_f_MI1_Override_Max_Speed :=120,

// Concrete Pump
_f_CP1_Max_Flowrate := INT_TO_REAL(GVL_RESD.n_Concrete_Pump_Max_Speed) * 
								   GVL_RESD.f_Concrete_Pump_dosing_volume,
_f_CP1_Check_Flowrate := GVL_RESD.f_Concrete_Pump_Check_Flowrate,
_t_CP1_Check_Duration := INT_TO_TIME(GVL_RESD.n_Concrete_Pump_Check_Duration*1000),

// Admixture pump (High)
_n_AP1_Max_Flowrate := GVL_RESD.n_Admixture_Pump_Max_Flowrate,
_n_AP1_Check_Flowrate := GVL_RESD.f_Admixture_Pump_Check_Flowrate,
_t_AP1_Check_Duration := INT_TO_TIME(GVL_RESD.n_Admixture_Pump_Check_Duration*1000),
_n_AP1_Flush_Flowrate := GVL_RESD.f_Admixture_Pump_Flush_Flowrate,
//_f_AP1_Check_Mass : REAL;

// Admixture pump (low)
_n_SP1_Max_Flowrate := GVL_RESD.n_Sup_Admixture_Pump_Max_Flowrate,
_n_SP1_Check_Flowrate := GVL_RESD.f_Sup_Admixture_Pump_Check_Flowrate,
_t_SP1_Check_Duration := INT_TO_TIME(GVL_RESD.n_Sup_Admixture_Pump_Check_Duration*1000),
//_f_SP1_Check_Mass : REAL;
);

//***********************************************************************************
// Setup IO data to PLC
//***********************************************************************************	
fb_SetOutputDataToIO(		
	// Mixer 
	b_MI1_set_run := GVL_ROB.ib_MI1_set_run,
	b_Ml1_Enable := GVL_ROB.ib_MI1_enable,
	b_MI1_Curved_Speed_On := GVL_ROB.ib_MI1_set_curved_speed_mode_on,
	f_MI1_Override_Speed := UINT_TO_REAL(GVL_ROB.in_MI1_set_speed),
	
	f_MI1_Override_Max_Speed := GVL_RESD.f_MI1_Override_Max_Speed,
	
	// Concrete Pump
	b_CP1_Forward_On := GVL_ROB.ib_CP1_forward_on,
	b_CP1_Backward_On := GVL_ROB.ib_CP1_backward_on,
	b_CP1_Flush_On := GVL_ROB.ib_CP1_flush_on,
	b_CP1_Check_On := GVL_ROB.ib_CP1_check_on,
	n_CP_Flowrate_mode := TRUE,
	n_CP1_Operate_Flowrate := REAL_TO_UDINT((UINT_TO_REAL(GVL_ROB.in_CP1_set_flowrate*10))),
	n_CP1_Check_Flowrate := REAL_TO_UDINT((UINT_TO_REAL(GVL_ROB.in_CP1_set_check_Flowrate*10))),
	n_CP1_Flush_Flowrate := REAL_TO_UDINT((UINT_TO_REAL(GVL_ROB.in_CP1_set_flush_flowrate*10))),
	f_dosing_volume := UINT_TO_INT(GVL_ROB.in_CP1_set_dosing_volume),
	
